LIN {X 0,Y 291.484,Z 681.746,A -85,B 0,C 180,E1 17047.292,E2 17047.292} C_VEL
LIN {X 0,Y 289.004,Z 660.075,A -85,B 0,C 180,E1 17052.26,E2 17052.26} C_VEL
LIN {X 0,Y 282.75,Z 637.12,A -85,B 0,C 180,E1 17057.64,E2 17057.64} C_VEL
LIN {X 0,Y 273.283,Z 615.443,A -85,B 0,C 180,E1 17063.436,E2 17063.436} C_VEL
LIN {X 0,Y 264.026,Z 599.669,A -85,B 0,C 180,E1 17068.648,E2 17068.648} C_VEL
LIN {X 0,Y 259.999,Z 593.567,A -85,B 0,C 180,E1 17071.016,E2 17071.016} C_VEL
LIN {X 0,Y 256.449,Z 587.64,A -85,B 0,C 180,E1 17073.314,E2 17073.314} C_VEL
LIN {X 0,Y 252.817,Z 583.048,A -85,B 0,C 180,E1 17075.688,E2 17075.688} C_VEL
LIN {X 0,Y 252.498,Z 580.66,A -85,B 0,C 180,E1 17076.137,E2 17076.137} C_VEL
LIN {X 0,Y 252.926,Z 580.66,A -85,B 0,C 180,E1 17083.299,E2 17083.299} C_VEL
LIN {X 0,Y 253.73,Z 580.66,A -85,B 0,C 180,E1 17093.136,E2 17093.136} C_VEL
LIN {X 0,Y 254.478,Z 580.66,A -85,B 0,C 180,E1 17099.99,E2 17099.99} C_VEL
LIN {X 0,Y 253.769,Z 580.66,A -85,B 0,C 180,E1 17106.843,E2 17106.843} C_VEL
LIN {X 0,Y 253.149,Z 580.66,A -85,B 0,C 180,E1 17113.831,E2 17113.831} C_VEL
LIN {X 0,Y 252.816,Z 580.66,A -85,B 0,C 180,E1 17117.976,E2 17117.976} C_VEL
LIN {X 0,Y 254.454,Z 585.604,A -85,B 0,C 180,E1 17119.318,E2 17119.318} C_VEL
LIN {X 0,Y 258.108,Z 589.393,A -85,B 0,C 180,E1 17121.472,E2 17121.472} C_VEL
LIN {X 0,Y 268.336,Z 604.22,A -85,B 0,C 180,E1 17126.709,E2 17126.709} C_VEL
LIN {X 0,Y 281.648,Z 625.679,A -85,B 0,C 180,E1 17132.393,E2 17132.393} C_VEL
LIN {X 0,Y 293.764,Z 651.604,A -85,B 0,C 180,E1 17137.493,E2 17137.493} C_VEL
LIN {X 0,Y 302.264,Z 679.148,A -85,B 0,C 180,E1 17141.931,E2 17141.931} C_VEL
LIN {X 0,Y 292.999,Z 713.963,A -85,B 0,C 180,E1 17144.982,E2 17144.982} C_VEL
LIN {X 0,Y 282.558,Z 745.546,A -85,B 0,C 180,E1 17149.094,E2 17149.094} C_VEL
LIN {X 0,Y 272.431,Z 773.196,A -85,B 0,C 180,E1 17154.352,E2 17154.352} C_VEL
LIN {X 0,Y 264.031,Z 796.979,A -85,B 0,C 180,E1 17160.826,E2 17160.826} C_VEL
LIN {X 0,Y 258.28,Z 816.418,A -85,B 0,C 180,E1 17168.505,E2 17168.505} C_VEL
LIN {X 0,Y 256.334,Z 829.468,A -85,B 0,C 180,E1 17176.331,E2 17176.331} C_VEL
LIN {X 0,Y 256.467,Z 836.245,A -85,B 0,C 180,E1 17183.216,E2 17183.216} C_VEL
LIN {X 0,Y 256.973,Z 838.591,A -85,B 0,C 180,E1 17189.997,E2 17189.997} C_VEL
LIN {X 0,Y 256.471,Z 836.262,A -85,B 0,C 180,E1 17196.777,E2 17196.777} C_VEL
LIN {X 0,Y 256.43,Z 828.378,A -85,B 0,C 180,E1 17204.529,E2 17204.529} C_VEL
LIN {X 0,Y 258.845,Z 814.689,A -85,B 0,C 180,E1 17212.342,E2 17212.342} C_VEL
LIN {X 0,Y 264.923,Z 794.449,A -85,B 0,C 180,E1 17220,E2 17220} C_VEL
LIN {X 0,Y 273.864,Z 769.676,A -85,B 0,C 180,E1 17226.456,E2 17226.456} C_VEL
LIN {X 0,Y 284.359,Z 740.416,A -85,B 0,C 180,E1 17231.705,E2 17231.705} C_VEL
LIN {X 0,Y 294.985,Z 707.872,A -85,B 0,C 180,E1 17235.668,E2 17235.668} C_VEL
LIN {X 0,Y 302.325,Z 679.287,A -85,B 0,C 180,E1 17238.079,E2 17238.079} C_VEL
LIN {X 0,Y 293.689,Z 651.111,A -85,B 0,C 180,E1 17242.612,E2 17242.612} C_VEL
LIN {X 0,Y 281.361,Z 624.993,A -85,B 0,C 180,E1 17247.798,E2 17247.798} C_VEL
LIN {X 0,Y 266.547,Z 601.233,A -85,B 0,C 180,E1 17254.232,E2 17254.232} C_VEL
LIN {X 0,Y 260.669,Z 593.537,A -85,B 0,C 180,E1 17257.169,E2 17257.169} C_VEL
LIN {X 0,Y 257.32,Z 587.873,A -85,B 0,C 180,E1 17259.141,E2 17259.141} C_VEL
LIN {X 0,Y 248.734,Z 587.348,A -85,B 0,C 180,E1 17264.144,E2 17264.144} C_VEL
LIN {X 0,Y 245.41,Z 582.419,A -85,B 0,C 180,E1 17267.087,E2 17267.087} C_VEL
LIN {X 0,Y 245.226,Z 580.66,A -85,B 0,C 180,E1 17267.531,E2 17267.531} C_VEL
LIN {X 0,Y 246.174,Z 580.66,A -85,B 0,C 180,E1 17276.484,E2 17276.484} C_VEL
LIN {X 0,Y 246.571,Z 580.66,A -85,B 0,C 180,E1 17280.01,E2 17280.01} C_VEL
LIN {X 0,Y 245.547,Z 580.66,A -85,B 0,C 180,E1 17289.43,E2 17289.43} C_VEL
LIN {X 0,Y 244.844,Z 580.933,A -85,B 0,C 180,E1 17298.253,E2 17298.253} C_VEL
LIN {X 0,Y 246.48,Z 585.654,A -85,B 0,C 180,E1 17300.107,E2 17300.107} C_VEL
LIN {X 0,Y 250.248,Z 588.949,A -85,B 0,C 180,E1 17303.05,E2 17303.05} C_VEL
LIN {X 0,Y 253.602,Z 594.604,A -85,B 0,C 180,E1 17305.659,E2 17305.659} C_VEL
LIN {X 0,Y 260.13,Z 605.185,A -85,B 0,C 180,E1 17310.114,E2 17310.114} C_VEL
LIN {X 0,Y 268.683,Z 620.445,A -85,B 0,C 180,E1 17315.49,E2 17315.49} C_VEL
LIN {X 0,Y 277.671,Z 642.456,A -85,B 0,C 180,E1 17321.657,E2 17321.657} C_VEL
LIN {X 0,Y 283.118,Z 664.136,A -85,B 0,C 180,E1 17327.005,E2 17327.005} C_VEL
LIN {X 0,Y 284.976,Z 686.052,A -85,B 0,C 180,E1 17332.261,E2 17332.261} C_VEL
LIN {X 0,Y 282.565,Z 694.344,A -85,B 0,C 180,E1 17333.89,E2 17333.89} C_VEL
LIN {X 0,Y 272.426,Z 717.171,A -85,B 0,C 180,E1 17339.068,E2 17339.068} C_VEL
LIN {X 0,Y 263.2,Z 735.869,A -85,B 0,C 180,E1 17345.355,E2 17345.355} C_VEL
LIN {X 0,Y 255.905,Z 749.866,A -85,B 0,C 180,E1 17352.797,E2 17352.797} C_VEL
LIN {X 0,Y 252.105,Z 757.453,A -85,B 0,C 180,E1 17359.624,E2 17359.624} C_VEL
LIN {X 0,Y 250.5,Z 761.052,A -85,B 0,C 180,E1 17366.538,E2 17366.538} C_VEL
LIN {X 0,Y 250.561,Z 761.007,A -85,B 0,C 180,E1 17373.467,E2 17373.467} C_VEL
LIN {X 0,Y 252.885,Z 755.837,A -85,B 0,C 180,E1 17382.099,E2 17382.099} C_VEL
LIN {X 0,Y 258.292,Z 745.196,A -85,B 0,C 180,E1 17390.003,E2 17390.003} C_VEL
LIN {X 0,Y 266.486,Z 729.264,A -85,B 0,C 180,E1 17397.037,E2 17397.037} C_VEL
LIN {X 0,Y 276.708,Z 707.849,A -85,B 0,C 180,E1 17403.175,E2 17403.175} C_VEL
LIN {X 0,Y 284.948,Z 687.938,A -85,B 0,C 180,E1 17407.141,E2 17407.141} C_VEL
LIN {X 0,Y 283.223,Z 665.7,A -85,B 0,C 180,E1 17412.51,E2 17412.51} C_VEL
LIN {X 0,Y 278.054,Z 643.824,A -85,B 0,C 180,E1 17417.844,E2 17417.844} C_VEL
LIN {X 0,Y 269.633,Z 622.585,A -85,B 0,C 180,E1 17423.715,E2 17423.715} C_VEL
LIN {X 0,Y 260.505,Z 605.867,A -85,B 0,C 180,E1 17429.442,E2 17429.442} C_VEL
LIN {X 0,Y 253.604,Z 594.637,A -85,B 0,C 180,E1 17434.104,E2 17434.104} C_VEL
LIN {X 0,Y 250.213,Z 589.003,A -85,B 0,C 180,E1 17436.711,E2 17436.711} C_VEL
LIN {X 0,Y 245.039,Z 582.819,A -85,B 0,C 180,E1 17441.061,E2 17441.061} C_VEL
LIN {X 0,Y 244.819,Z 580.66,A -85,B 0,C 180,E1 17441.745,E2 17441.745} C_VEL
LIN {X 0,Y 245.509,Z 580.66,A -85,B 0,C 180,E1 17450.663,E2 17450.663} C_VEL
LIN {X 0,Y 246.202,Z 580.66,A -85,B 0,C 180,E1 17456.465,E2 17456.465} C_VEL
LIN {X 0,Y 246.568,Z 580.66,A -85,B 0,C 180,E1 17459.99,E2 17459.99} C_VEL
LIN {X 0,Y 245.554,Z 580.66,A -85,B 0,C 180,E1 17469.4,E2 17469.4} C_VEL
LIN {X 0,Y 245.295,Z 581.397,A -85,B 0,C 180,E1 17472.919,E2 17472.919} C_VEL
LIN {X 0,Y 247.819,Z 586.604,A -85,B 0,C 180,E1 17475.335,E2 17475.335} C_VEL
LIN {X 0,Y 250.708,Z 589.38,A -85,B 0,C 180,E1 17477.455,E2 17477.455} C_VEL
LIN {X 0,Y 254.799,Z 594.985,A -85,B 0,C 180,E1 17480.195,E2 17480.195} C_VEL
LIN {X 0,Y 265.726,Z 611.439,A -85,B 0,C 180,E1 17486.194,E2 17486.194} C_VEL
LIN {X 0,Y 277.92,Z 632.265,A -85,B 0,C 180,E1 17491.843,E2 17491.843} C_VEL
LIN {X 0,Y 288.974,Z 657.419,A -85,B 0,C 180,E1 17496.988,E2 17496.988} C_VEL
LIN {X 0,Y 295.98,Z 681.869,A -85,B 0,C 180,E1 17501.112,E2 17501.112} C_VEL
LIN {X 0,Y 285.816,Z 717.211,A -85,B 0,C 180,E1 17504.343,E2 17504.343} C_VEL
LIN {X 0,Y 274.522,Z 749.194,A -85,B 0,C 180,E1 17508.821,E2 17508.821} C_VEL
LIN {X 0,Y 263.808,Z 777.218,A -85,B 0,C 180,E1 17514.59,E2 17514.59} C_VEL
LIN {X 0,Y 255.114,Z 800.615,A -85,B 0,C 180,E1 17521.652,E2 17521.652} C_VEL
LIN {X 0,Y 249.861,Z 818.715,A -85,B 0,C 180,E1 17529.658,E2 17529.658} C_VEL
LIN {X 0,Y 248.446,Z 829.786,A -85,B 0,C 180,E1 17537.128,E2 17537.128} C_VEL
LIN {X 0,Y 248.614,Z 835.043,A -85,B 0,C 180,E1 17543.001,E2 17543.001} C_VEL
LIN {X 0,Y 249.15,Z 837.403,A -85,B 0,C 180,E1 17549.997,E2 17549.997} C_VEL
LIN {X 0,Y 248.62,Z 835.06,A -85,B 0,C 180,E1 17556.992,E2 17556.992} C_VEL
LIN {X 0,Y 248.614,Z 827.147,A -85,B 0,C 180,E1 17564.997,E2 17564.997} C_VEL
LIN {X 0,Y 251.283,Z 813.429,A -85,B 0,C 180,E1 17573.053,E2 17573.053} C_VEL
LIN {X 0,Y 257.823,Z 793.166,A -85,B 0,C 180,E1 17580.915,E2 17580.915} C_VEL
LIN {X 0,Y 267.53,Z 767.817,A -85,B 0,C 180,E1 17587.614,E2 17587.614} C_VEL
LIN {X 0,Y 278.305,Z 739.048,A -85,B 0,C 180,E1 17592.825,E2 17592.825} C_VEL
LIN {X 0,Y 289.404,Z 706.392,A -85,B 0,C 180,E1 17596.81,E2 17596.81} C_VEL
LIN {X 0,Y 295.831,Z 680.996,A -85,B 0,C 180,E1 17599.06,E2 17599.06} C_VEL
LIN {X 0,Y 287.805,Z 654.157,A -85,B 0,C 180,E1 17603.663,E2 17603.663} C_VEL
LIN {X 0,Y 276.684,Z 629.753,A -85,B 0,C 180,E1 17608.803,E2 17608.803} C_VEL
LIN {X 0,Y 263.656,Z 607.901,A -85,B 0,C 180,E1 17614.954,E2 17614.954} C_VEL
LIN {X 0,Y 254.144,Z 594.536,A -85,B 0,C 180,E1 17620.318,E2 17620.318} C_VEL
LIN {X 0,Y 250.515,Z 588.746,A -85,B 0,C 180,E1 17622.875,E2 17622.875} C_VEL
LIN {X 0,Y 248.734,Z 587.348,A -85,B 0,C 180,E1 17624.144,E2 17624.144} C_VEL
LIN {X 0,Y 242.06,Z 587.782,A -85,B 0,C 180,E1 17629.455,E2 17629.455} C_VEL
LIN {X 0,Y 238.235,Z 582.554,A -85,B 0,C 180,E1 17635.111,E2 17635.111} C_VEL
LIN {X 0,Y 238.155,Z 580.66,A -85,B 0,C 180,E1 17635.909,E2 17635.909} C_VEL
LIN {X 0,Y 238.66,Z 580.66,A -85,B 0,C 180,E1 17640.01,E2 17640.01} C_VEL
LIN {X 0,Y 237.666,Z 581.2,A -85,B 0,C 180,E1 17649.443,E2 17649.443} C_VEL
LIN {X 0,Y 239.854,Z 586.504,A -85,B 0,C 180,E1 17653.936,E2 17653.936} C_VEL
LIN {X 0,Y 243.016,Z 589.19,A -85,B 0,C 180,E1 17657.679,E2 17657.679} C_VEL
LIN {X 0,Y 246.273,Z 594.62,A -85,B 0,C 180,E1 17661.044,E2 17661.044} C_VEL
LIN {X 0,Y 248.141,Z 596.956,A -85,B 0,C 180,E1 17662.664,E2 17662.664} C_VEL
LIN {X 0,Y 256.047,Z 609.94,A -85,B 0,C 180,E1 17668.846,E2 17668.846} C_VEL
LIN {X 0,Y 265.703,Z 629.267,A -85,B 0,C 180,E1 17675.749,E2 17675.749} C_VEL
LIN {X 0,Y 273.446,Z 651.309,A -85,B 0,C 180,E1 17682.026,E2 17682.026} C_VEL
LIN {X 0,Y 277.677,Z 672.925,A -85,B 0,C 180,E1 17687.564,E2 17687.564} C_VEL
LIN {X 0,Y 277.956,Z 691.579,A -85,B 0,C 180,E1 17692.207,E2 17692.207} C_VEL
LIN {X 0,Y 267.183,Z 715.618,A -85,B 0,C 180,E1 17697.434,E2 17697.434} C_VEL
LIN {X 0,Y 257.196,Z 735.039,A -85,B 0,C 180,E1 17703.804,E2 17703.804} C_VEL
LIN {X 0,Y 249.54,Z 749.077,A -85,B 0,C 180,E1 17710.885,E2 17710.885} C_VEL
LIN {X 0,Y 244.43,Z 758.639,A -85,B 0,C 180,E1 17719.294,E2 17719.294} C_VEL
LIN {X 0,Y 242.708,Z 762.238,A -85,B 0,C 180,E1 17726.427,E2 17726.427} C_VEL
LIN {X 0,Y 242.76,Z 762.195,A -85,B 0,C 180,E1 17733.579,E2 17733.579} C_VEL
LIN {X 0,Y 245.265,Z 757.026,A -85,B 0,C 180,E1 17742.481,E2 17742.481} C_VEL
LIN {X 0,Y 250.964,Z 746.39,A -85,B 0,C 180,E1 17750.613,E2 17750.613} C_VEL
LIN {X 0,Y 259.539,Z 730.479,A -85,B 0,C 180,E1 17757.822,E2 17757.822} C_VEL
LIN {X 0,Y 270.224,Z 709.091,A -85,B 0,C 180,E1 17764.079,E2 17764.079} C_VEL
LIN {X 0,Y 278.32,Z 689.31,A -85,B 0,C 180,E1 17768.182,E2 17768.182} C_VEL
LIN {X 0,Y 276.857,Z 667.842,A -85,B 0,C 180,E1 17773.59,E2 17773.59} C_VEL
LIN {X 0,Y 271.994,Z 646.383,A -85,B 0,C 180,E1 17779.127,E2 17779.127} C_VEL
LIN {X 0,Y 264.392,Z 626.168,A -85,B 0,C 180,E1 17785.054,E2 17785.054} C_VEL
LIN {X 0,Y 254.755,Z 607.962,A -85,B 0,C 180,E1 17791.849,E2 17791.849} C_VEL
LIN {X 0,Y 250.273,Z 600.944,A -85,B 0,C 180,E1 17795.247,E2 17795.247} C_VEL
LIN {X 0,Y 246.888,Z 595.127,A -85,B 0,C 180,E1 17798.164,E2 17798.164} C_VEL
LIN {X 0,Y 243.091,Z 589.722,A -85,B 0,C 180,E1 17801.845,E2 17801.845} C_VEL
LIN {X 0,Y 242.171,Z 588.089,A -85,B 0,C 180,E1 17802.907,E2 17802.907} C_VEL
LIN {X 0,Y 237.857,Z 583.161,A -85,B 0,C 180,E1 17809.067,E2 17809.067} C_VEL
LIN {X 0,Y 237.594,Z 580.66,A -85,B 0,C 180,E1 17810.349,E2 17810.349} C_VEL
LIN {X 0,Y 238.273,Z 580.66,A -85,B 0,C 180,E1 17816.347,E2 17816.347} C_VEL
LIN {X 0,Y 238.657,Z 580.66,A -85,B 0,C 180,E1 17819.99,E2 17819.99} C_VEL
LIN {X 0,Y 238.09,Z 581.405,A -85,B 0,C 180,E1 17824.892,E2 17824.892} C_VEL
LIN {X 0,Y 240.232,Z 586.467,A -85,B 0,C 180,E1 17828.716,E2 17828.716} C_VEL
LIN {X 0,Y 243.552,Z 589.301,A -85,B 0,C 180,E1 17832.329,E2 17832.329} C_VEL
LIN {X 0,Y 247.027,Z 594.819,A -85,B 0,C 180,E1 17835.544,E2 17835.544} C_VEL
LIN {X 0,Y 248.92,Z 597.304,A -85,B 0,C 180,E1 17837.01,E2 17837.01} C_VEL
LIN {X 0,Y 254.727,Z 605.939,A -85,B 0,C 180,E1 17840.997,E2 17840.997} C_VEL
LIN {X 0,Y 263.523,Z 619.355,A -85,B 0,C 180,E1 17845.971,E2 17845.971} C_VEL
LIN {X 0,Y 275.76,Z 642.16,A -85,B 0,C 180,E1 17852.122,E2 17852.122} C_VEL
LIN {X 0,Y 285.4,Z 667.461,A -85,B 0,C 180,E1 17857.271,E2 17857.271} C_VEL
LIN {X 0,Y 289.633,Z 684.994,A -85,B 0,C 180,E1 17860.282,E2 17860.282} C_VEL
LIN {X 0,Y 278.654,Z 720.111,A -85,B 0,C 180,E1 17863.667,E2 17863.667} C_VEL
LIN {X 0,Y 267.152,Z 751.162,A -85,B 0,C 180,E1 17868.244,E2 17868.244} C_VEL
LIN {X 0,Y 255.963,Z 778.674,A -85,B 0,C 180,E1 17874.256,E2 17874.256} C_VEL
LIN {X 0,Y 247.441,Z 800.68,A -85,B 0,C 180,E1 17881.252,E2 17881.252} C_VEL
LIN {X 0,Y 241.917,Z 818.856,A -85,B 0,C 180,E1 17889.817,E2 17889.817} C_VEL
LIN {X 0,Y 240.556,Z 829.8,A -85,B 0,C 180,E1 17897.908,E2 17897.908} C_VEL
LIN {X 0,Y 240.76,Z 833.839,A -85,B 0,C 180,E1 17902.771,E2 17902.771} C_VEL
LIN {X 0,Y 241.326,Z 836.214,A -85,B 0,C 180,E1 17909.997,E2 17909.997} C_VEL
LIN {X 0,Y 240.766,Z 833.858,A -85,B 0,C 180,E1 17917.222,E2 17917.222} C_VEL
LIN {X 0,Y 240.804,Z 825.915,A -85,B 0,C 180,E1 17925.495,E2 17925.495} C_VEL
LIN {X 0,Y 243.72,Z 812.161,A -85,B 0,C 180,E1 17933.812,E2 17933.812} C_VEL
LIN {X 0,Y 250.713,Z 792.046,A -85,B 0,C 180,E1 17941.83,E2 17941.83} C_VEL
LIN {X 0,Y 261.116,Z 766.508,A -85,B 0,C 180,E1 17948.706,E2 17948.706} C_VEL
LIN {X 0,Y 272.271,Z 737.882,A -85,B 0,C 180,E1 17953.966,E2 17953.966} C_VEL
LIN {X 0,Y 283.902,Z 704.895,A -85,B 0,C 180,E1 17958.007,E2 17958.007} C_VEL
LIN {X 0,Y 289.587,Z 683.6,A -85,B 0,C 180,E1 17959.943,E2 17959.943} C_VEL
LIN {X 0,Y 282.141,Z 657.535,A -85,B 0,C 180,E1 17964.653,E2 17964.653} C_VEL
LIN {X 0,Y 271.947,Z 634.447,A -85,B 0,C 180,E1 17969.825,E2 17969.825} C_VEL
LIN {X 0,Y 260.53,Z 614.345,A -85,B 0,C 180,E1 17975.779,E2 17975.779} C_VEL
LIN {X 0,Y 251.677,Z 601.43,A -85,B 0,C 180,E1 17981.145,E2 17981.145} C_VEL
LIN {X 0,Y 247.246,Z 594.982,A -85,B 0,C 180,E1 17984.47,E2 17984.47} C_VEL
LIN {X 0,Y 243.547,Z 589.353,A -85,B 0,C 180,E1 17987.899,E2 17987.899} C_VEL
LIN {X 0,Y 242.06,Z 587.782,A -85,B 0,C 180,E1 17989.455,E2 17989.455} C_VEL
LIN {X 0,Y 236.289,Z 588.291,A -85,B 0,C 180,E1 17997.671,E2 17997.671} C_VEL
LIN {X 0,Y 236.476,Z 589.167,A -85,B 0,C 180,E1 18009.071,E2 18009.071} C_VEL
LIN {X 0,Y 239.066,Z 594.704,A -85,B 0,C 180,E1 18014.45,E2 18014.45} C_VEL
LIN {X 0,Y 241.246,Z 597.021,A -85,B 0,C 180,E1 18017.26,E2 18017.26} C_VEL
LIN {X 0,Y 244.913,Z 602.642,A -85,B 0,C 180,E1 18021.232,E2 18021.232} C_VEL
LIN {X 0,Y 252.764,Z 616.714,A -85,B 0,C 180,E1 18028.277,E2 18028.277} C_VEL
LIN {X 0,Y 261.635,Z 635.872,A -85,B 0,C 180,E1 18035.369,E2 18035.369} C_VEL
LIN {X 0,Y 268.096,Z 656.605,A -85,B 0,C 180,E1 18041.522,E2 18041.522} C_VEL
LIN {X 0,Y 271.517,Z 677.591,A -85,B 0,C 180,E1 18047.151,E2 18047.151} C_VEL
LIN {X 0,Y 271.508,Z 693.613,A -85,B 0,C 180,E1 18051.338,E2 18051.338} C_VEL
LIN {X 0,Y 259.89,Z 718.23,A -85,B 0,C 180,E1 18056.9,E2 18056.9} C_VEL
LIN {X 0,Y 249.089,Z 738.273,A -85,B 0,C 180,E1 18063.857,E2 18063.857} C_VEL
LIN {X 0,Y 240.981,Z 752.253,A -85,B 0,C 180,E1 18071.695,E2 18071.695} C_VEL
LIN {X 0,Y 236.751,Z 759.827,A -85,B 0,C 180,E1 18078.943,E2 18078.943} C_VEL
LIN {X 0,Y 234.93,Z 763.421,A -85,B 0,C 180,E1 18086.308,E2 18086.308} C_VEL
LIN {X 0,Y 234.981,Z 763.379,A -85,B 0,C 180,E1 18093.698,E2 18093.698} C_VEL
LIN {X 0,Y 237.624,Z 758.219,A -85,B 0,C 180,E1 18102.889,E2 18102.889} C_VEL
LIN {X 0,Y 243.553,Z 747.763,A -85,B 0,C 180,E1 18111.151,E2 18111.151} C_VEL
LIN {X 0,Y 252.664,Z 731.689,A -85,B 0,C 180,E1 18118.648,E2 18118.648} C_VEL
LIN {X 0,Y 263.805,Z 710.331,A -85,B 0,C 180,E1 18125.028,E2 18125.028} C_VEL
LIN {X 0,Y 271.698,Z 692.758,A -85,B 0,C 180,E1 18128.712,E2 18128.712} C_VEL
LIN {X 0,Y 270.897,Z 672.694,A -85,B 0,C 180,E1 18134.023,E2 18134.023} C_VEL
LIN {X 0,Y 266.687,Z 651.162,A -85,B 0,C 180,E1 18139.858,E2 18139.858} C_VEL
LIN {X 0,Y 260.015,Z 631.997,A -85,B 0,C 180,E1 18145.728,E2 18145.728} C_VEL
LIN {X 0,Y 251.413,Z 614.593,A -85,B 0,C 180,E1 18152.533,E2 18152.533} C_VEL
LIN {X 0,Y 246.97,Z 607.143,A -85,B 0,C 180,E1 18156.315,E2 18156.315} C_VEL
LIN {X 0,Y 244.314,Z 602.206,A -85,B 0,C 180,E1 18158.992,E2 18158.992} C_VEL
LIN {X 0,Y 240.973,Z 596.177,A -85,B 0,C 180,E1 18162.801,E2 18162.801} C_VEL
LIN {X 0,Y 236.532,Z 590.526,A -85,B 0,C 180,E1 18169.674,E2 18169.674} C_VEL
LIN {X 0,Y 236.148,Z 588.418,A -85,B 0,C 180,E1 18171.167,E2 18171.167} C_VEL
LIN {X 0,Y 236.756,Z 588.624,A -85,B 0,C 180,E1 18184.115,E2 18184.115} C_VEL
LIN {X 0,Y 239.158,Z 594.317,A -85,B 0,C 180,E1 18188.637,E2 18188.637} C_VEL
LIN {X 0,Y 241.971,Z 597.044,A -85,B 0,C 180,E1 18191.837,E2 18191.837} C_VEL
LIN {X 0,Y 245.968,Z 602.77,A -85,B 0,C 180,E1 18195.612,E2 18195.612} C_VEL
LIN {X 0,Y 255.448,Z 617.73,A -85,B 0,C 180,E1 18202.419,E2 18202.419} C_VEL
LIN {X 0,Y 266.117,Z 636.709,A -85,B 0,C 180,E1 18208.561,E2 18208.561} C_VEL
LIN {X 0,Y 275.962,Z 659.496,A -85,B 0,C 180,E1 18214.058,E2 18214.058} C_VEL
LIN {X 0,Y 283.36,Z 686.138,A -85,B 0,C 180,E1 18219.182,E2 18219.182} C_VEL
LIN {X 0,Y 272.532,Z 720.298,A -85,B 0,C 180,E1 18222.63,E2 18222.63} C_VEL
LIN {X 0,Y 260.217,Z 751.913,A -85,B 0,C 180,E1 18227.435,E2 18227.435} C_VEL
LIN {X 0,Y 248.678,Z 778.946,A -85,B 0,C 180,E1 18233.583,E2 18233.583} C_VEL
LIN {X 0,Y 239.535,Z 801.306,A -85,B 0,C 180,E1 18241.051,E2 18241.051} C_VEL
LIN {X 0,Y 234.224,Z 817.599,A -85,B 0,C 180,E1 18249.123,E2 18249.123} C_VEL
LIN {X 0,Y 232.69,Z 828.457,A -85,B 0,C 180,E1 18257.373,E2 18257.373} C_VEL
LIN {X 0,Y 232.906,Z 832.636,A -85,B 0,C 180,E1 18262.526,E2 18262.526} C_VEL
LIN {X 0,Y 233.501,Z 835.026,A -85,B 0,C 180,E1 18269.997,E2 18269.997} C_VEL
LIN {X 0,Y 232.914,Z 832.656,A -85,B 0,C 180,E1 18277.467,E2 18277.467} C_VEL
LIN {X 0,Y 233.013,Z 824.682,A -85,B 0,C 180,E1 18286.027,E2 18286.027} C_VEL
LIN {X 0,Y 236.213,Z 810.896,A -85,B 0,C 180,E1 18294.618,E2 18294.618} C_VEL
LIN {X 0,Y 243.79,Z 790.821,A -85,B 0,C 180,E1 18302.828,E2 18302.828} C_VEL
LIN {X 0,Y 254.627,Z 765.428,A -85,B 0,C 180,E1 18309.813,E2 18309.813} C_VEL
LIN {X 0,Y 266.467,Z 736.529,A -85,B 0,C 180,E1 18315.181,E2 18315.181} C_VEL
LIN {X 0,Y 278.26,Z 704.396,A -85,B 0,C 180,E1 18319.146,E2 18319.146} C_VEL
LIN {X 0,Y 283.398,Z 686.418,A -85,B 0,C 180,E1 18320.816,E2 18320.816} C_VEL
LIN {X 0,Y 276.553,Z 660.888,A -85,B 0,C 180,E1 18325.689,E2 18325.689} C_VEL
LIN {X 0,Y 266.944,Z 638.252,A -85,B 0,C 180,E1 18331.072,E2 18331.072} C_VEL
LIN {X 0,Y 256.73,Z 619.872,A -85,B 0,C 180,E1 18336.897,E2 18336.897} C_VEL
LIN {X 0,Y 249.144,Z 608.232,A -85,B 0,C 180,E1 18341.979,E2 18341.979} C_VEL
LIN {X 0,Y 245.37,Z 602.346,A -85,B 0,C 180,E1 18345.036,E2 18345.036} C_VEL
LIN {X 0,Y 241.741,Z 596.221,A -85,B 0,C 180,E1 18348.723,E2 18348.723} C_VEL
LIN {X 0,Y 237.07,Z 590.392,A -85,B 0,C 180,E1 18355.431,E2 18355.431} C_VEL
LIN {X 0,Y 236.448,Z 588.331,A -85,B 0,C 180,E1 18357.258,E2 18357.258} C_VEL
LIN {X 0,Y 236.289,Z 588.291,A -85,B 0,C 180,E1 18357.671,E2 18357.671} C_VEL
LIN {X 0,Y 234.846,Z 591.965,A -85,B 0,C 180,E1 18361.814,E2 18361.814} C_VEL
LIN {X 0,Y 234.493,Z 596.014,A -85,B 0,C 180,E1 18365.988,E2 18365.988} C_VEL
LIN {X 0,Y 235.214,Z 597.29,A -85,B 0,C 180,E1 18368.902,E2 18368.902} C_VEL
LIN {X 0,Y 237.932,Z 602.797,A -85,B 0,C 180,E1 18374.951,E2 18374.951} C_VEL
LIN {X 0,Y 239.408,Z 605.1,A -85,B 0,C 180,E1 18377.049,E2 18377.049} C_VEL
LIN {X 0,Y 243.461,Z 612.242,A -85,B 0,C 180,E1 18381.919,E2 18381.919} C_VEL
LIN {X 0,Y 249.259,Z 623.12,A -85,B 0,C 180,E1 18387.602,E2 18387.602} C_VEL
LIN {X 0,Y 257.37,Z 642.395,A -85,B 0,C 180,E1 18395.01,E2 18395.01} C_VEL
LIN {X 0,Y 263.088,Z 663.82,A -85,B 0,C 180,E1 18401.576,E2 18401.576} C_VEL
LIN {X 0,Y 265.468,Z 684.446,A -85,B 0,C 180,E1 18407.344,E2 18407.344} C_VEL
LIN {X 0,Y 264.76,Z 696.526,A -85,B 0,C 180,E1 18410.594,E2 18410.594} C_VEL
LIN {X 0,Y 252.628,Z 720.834,A -85,B 0,C 180,E1 18416.337,E2 18416.337} C_VEL
LIN {X 0,Y 242.086,Z 739.476,A -85,B 0,C 180,E1 18423.04,E2 18423.04} C_VEL
LIN {X 0,Y 233.555,Z 753.447,A -85,B 0,C 180,E1 18431.091,E2 18431.091} C_VEL
LIN {X 0,Y 229.082,Z 761.015,A -85,B 0,C 180,E1 18438.568,E2 18438.568} C_VEL
LIN {X 0,Y 227.158,Z 764.604,A -85,B 0,C 180,E1 18446.182,E2 18446.182} C_VEL
LIN {X 0,Y 227.187,Z 764.566,A -85,B 0,C 180,E1 18453.825,E2 18453.825} C_VEL
LIN {X 0,Y 230.007,Z 759.409,A -85,B 0,C 180,E1 18463.323,E2 18463.323} C_VEL
LIN {X 0,Y 236.265,Z 748.959,A -85,B 0,C 180,E1 18471.836,E2 18471.836} C_VEL
LIN {X 0,Y 245.824,Z 732.904,A -85,B 0,C 180,E1 18479.523,E2 18479.523} C_VEL
LIN {X 0,Y 257.452,Z 711.57,A -85,B 0,C 180,E1 18486.025,E2 18486.025} C_VEL
LIN {X 0,Y 265.19,Z 694.135,A -85,B 0,C 180,E1 18489.848,E2 18489.848} C_VEL
LIN {X 0,Y 264.585,Z 674.128,A -85,B 0,C 180,E1 18495.385,E2 18495.385} C_VEL
LIN {X 0,Y 260.672,Z 653.388,A -85,B 0,C 180,E1 18501.352,E2 18501.352} C_VEL
LIN {X 0,Y 254.264,Z 634.706,A -85,B 0,C 180,E1 18507.583,E2 18507.583} C_VEL
LIN {X 0,Y 245.938,Z 616.464,A -85,B 0,C 180,E1 18515.315,E2 18515.315} C_VEL
LIN {X 0,Y 241.539,Z 609.13,A -85,B 0,C 180,E1 18519.826,E2 18519.826} C_VEL
LIN {X 0,Y 238.359,Z 603.169,A -85,B 0,C 180,E1 18524.075,E2 18524.075} C_VEL
LIN {X 0,Y 235.103,Z 597.709,A -85,B 0,C 180,E1 18530.417,E2 18530.417} C_VEL
LIN {X 0,Y 234.697,Z 596.131,A -85,B 0,C 180,E1 18532.021,E2 18532.021} C_VEL
LIN {X 0,Y 235.482,Z 596.488,A -85,B 0,C 180,E1 18543.676,E2 18543.676} C_VEL
LIN {X 0,Y 238.555,Z 602.693,A -85,B 0,C 180,E1 18549.349,E2 18549.349} C_VEL
LIN {X 0,Y 240.442,Z 605.051,A -85,B 0,C 180,E1 18551.568,E2 18551.568} C_VEL
LIN {X 0,Y 245.157,Z 612.751,A -85,B 0,C 180,E1 18556.24,E2 18556.24} C_VEL
LIN {X 0,Y 252.377,Z 624.173,A -85,B 0,C 180,E1 18561.663,E2 18561.663} C_VEL
LIN {X 0,Y 262.542,Z 643.595,A -85,B 0,C 180,E1 18568.141,E2 18568.141} C_VEL
LIN {X 0,Y 271.647,Z 666.876,A -85,B 0,C 180,E1 18573.862,E2 18573.862} C_VEL
LIN {X 0,Y 277.054,Z 688.498,A -85,B 0,C 180,E1 18578.198,E2 18578.198} C_VEL
LIN {X 0,Y 265.974,Z 721.928,A -85,B 0,C 180,E1 18581.723,E2 18581.723} C_VEL
LIN {X 0,Y 253.346,Z 752.61,A -85,B 0,C 180,E1 18586.583,E2 18586.583} C_VEL
LIN {X 0,Y 241.414,Z 779.216,A -85,B 0,C 180,E1 18592.866,E2 18592.866} C_VEL
LIN {X 0,Y 231.809,Z 801.392,A -85,B 0,C 180,E1 18600.665,E2 18600.665} C_VEL
LIN {X 0,Y 226.193,Z 818.129,A -85,B 0,C 180,E1 18609.539,E2 18609.539} C_VEL
LIN {X 0,Y 224.824,Z 828.563,A -85,B 0,C 180,E1 18618.341,E2 18618.341} C_VEL
LIN {X 0,Y 225.251,Z 833.15,A -85,B 0,C 180,E1 18626.142,E2 18626.142} C_VEL
LIN {X 0,Y 225.693,Z 833.839,A -85,B 0,C 180,E1 18629.996,E2 18629.996} C_VEL
LIN {X 0,Y 225.051,Z 831.45,A -85,B 0,C 180,E1 18637.729,E2 18637.729} C_VEL
LIN {X 0,Y 225.221,Z 823.447,A -85,B 0,C 180,E1 18646.597,E2 18646.597} C_VEL
LIN {X 0,Y 228.788,Z 809.639,A -85,B 0,C 180,E1 18655.473,E2 18655.473} C_VEL
LIN {X 0,Y 236.697,Z 789.969,A -85,B 0,C 180,E1 18663.761,E2 18663.761} C_VEL
LIN {X 0,Y 248.237,Z 764.362,A -85,B 0,C 180,E1 18670.975,E2 18670.975} C_VEL
LIN {X 0,Y 260.886,Z 734.892,A -85,B 0,C 180,E1 18676.497,E2 18676.497} C_VEL
LIN {X 0,Y 273.475,Z 701.54,A -85,B 0,C 180,E1 18680.563,E2 18680.563} C_VEL
LIN {X 0,Y 277.148,Z 688.614,A -85,B 0,C 180,E1 18681.814,E2 18681.814} C_VEL
LIN {X 0,Y 270.718,Z 663.708,A -85,B 0,C 180,E1 18686.872,E2 18686.872} C_VEL
LIN {X 0,Y 262.159,Z 642.794,A -85,B 0,C 180,E1 18692.172,E2 18692.172} C_VEL
LIN {X 0,Y 251.869,Z 622.901,A -85,B 0,C 180,E1 18698.869,E2 18698.869} C_VEL
LIN {X 0,Y 243.253,Z 609.621,A -85,B 0,C 180,E1 18705.709,E2 18705.709} C_VEL
LIN {X 0,Y 239.182,Z 603.072,A -85,B 0,C 180,E1 18710.215,E2 18710.215} C_VEL
LIN {X 0,Y 235.625,Z 597.118,A -85,B 0,C 180,E1 18716.441,E2 18716.441} C_VEL
LIN {X 0,Y 234.572,Z 595.791,A -85,B 0,C 180,E1 18720.01,E2 18720.01} C_VEL
LIN {X 0,Y 234.493,Z 596.014,A -85,B 0,C 180,E1 18725.988,E2 18725.988} C_VEL
LIN {X 0,Y 234.465,Z 599.493,A -85,B 0,C 180,E1 18727.941,E2 18727.941} C_VEL
LIN {X 0,Y 234.076,Z 607.442,A -85,B 0,C 180,E1 18730.656,E2 18730.656} C_VEL
LIN {X 0,Y 234.171,Z 607.839,A -85,B 0,C 180,E1 18731.011,E2 18731.011} C_VEL
LIN {X 0,Y 237.087,Z 612.234,A -85,B 0,C 180,E1 18736.451,E2 18736.451} C_VEL
LIN {X 0,Y 240.824,Z 619.853,A -85,B 0,C 180,E1 18741.652,E2 18741.652} C_VEL
LIN {X 0,Y 246.299,Z 631.438,A -85,B 0,C 180,E1 18747.693,E2 18747.693} C_VEL
LIN {X 0,Y 252.669,Z 648.009,A -85,B 0,C 180,E1 18754.335,E2 18754.335} C_VEL
LIN {X 0,Y 257.475,Z 668.445,A -85,B 0,C 180,E1 18760.902,E2 18760.902} C_VEL
LIN {X 0,Y 259.135,Z 687.764,A -85,B 0,C 180,E1 18766.587,E2 18766.587} C_VEL
LIN {X 0,Y 258.064,Z 699.358,A -85,B 0,C 180,E1 18769.812,E2 18769.812} C_VEL
LIN {X 0,Y 245.373,Z 723.442,A -85,B 0,C 180,E1 18775.738,E2 18775.738} C_VEL
LIN {X 0,Y 233.959,Z 742.504,A -85,B 0,C 180,E1 18783.068,E2 18783.068} C_VEL
LIN {X 0,Y 225.425,Z 755.866,A -85,B 0,C 180,E1 18791.4,E2 18791.4} C_VEL
LIN {X 0,Y 220.659,Z 763.46,A -85,B 0,C 180,E1 18800.127,E2 18800.127} C_VEL
LIN {X 0,Y 219.382,Z 765.788,A -85,B 0,C 180,E1 18806.046,E2 18806.046} C_VEL
LIN {X 0,Y 219.411,Z 765.75,A -85,B 0,C 180,E1 18813.96,E2 18813.96} C_VEL
LIN {X 0,Y 222.393,Z 760.602,A -85,B 0,C 180,E1 18823.788,E2 18823.788} C_VEL
LIN {X 0,Y 228.616,Z 750.793,A -85,B 0,C 180,E1 18832.144,E2 18832.144} C_VEL
LIN {X 0,Y 238.413,Z 735.245,A -85,B 0,C 180,E1 18840.01,E2 18840.01} C_VEL
LIN {X 0,Y 250.367,Z 714.322,A -85,B 0,C 180,E1 18846.671,E2 18846.671} C_VEL
LIN {X 0,Y 258.581,Z 697.735,A -85,B 0,C 180,E1 18850.418,E2 18850.418} C_VEL
LIN {X 0,Y 258.609,Z 678.667,A -85,B 0,C 180,E1 18855.936,E2 18855.936} C_VEL
LIN {X 0,Y 255.593,Z 659.173,A -85,B 0,C 180,E1 18861.797,E2 18861.797} C_VEL
LIN {X 0,Y 249.857,Z 640.253,A -85,B 0,C 180,E1 18868.389,E2 18868.389} C_VEL
LIN {X 0,Y 242.643,Z 623.152,A -85,B 0,C 180,E1 18876.061,E2 18876.061} C_VEL
LIN {X 0,Y 238.722,Z 615.994,A -85,B 0,C 180,E1 18880.659,E2 18880.659} C_VEL
LIN {X 0,Y 235.952,Z 610.472,A -85,B 0,C 180,E1 18884.903,E2 18884.903} C_VEL
LIN {X 0,Y 233.428,Z 604.81,A -85,B 0,C 180,E1 18891.158,E2 18891.158} C_VEL
LIN {X 0,Y 232.644,Z 603.485,A -85,B 0,C 180,E1 18896.258,E2 18896.258} C_VEL
LIN {X 0,Y 234.14,Z 604.781,A -85,B 0,C 180,E1 18903.581,E2 18903.581} C_VEL
LIN {X 0,Y 237.496,Z 610.705,A -85,B 0,C 180,E1 18909.746,E2 18909.746} C_VEL
LIN {X 0,Y 243.052,Z 620.424,A -85,B 0,C 180,E1 18915.92,E2 18915.92} C_VEL
LIN {X 0,Y 249.801,Z 631.987,A -85,B 0,C 180,E1 18921.431,E2 18921.431} C_VEL
LIN {X 0,Y 258.459,Z 649.681,A -85,B 0,C 180,E1 18927.49,E2 18927.49} C_VEL
LIN {X 0,Y 266.518,Z 671.969,A -85,B 0,C 180,E1 18933.183,E2 18933.183} C_VEL
LIN {X 0,Y 270.814,Z 692.585,A -85,B 0,C 180,E1 18937.43,E2 18937.43} C_VEL
LIN {X 0,Y 258.577,Z 725.604,A -85,B 0,C 180,E1 18941.07,E2 18941.07} C_VEL
LIN {X 0,Y 245.55,Z 755.455,A -85,B 0,C 180,E1 18946.112,E2 18946.112} C_VEL
LIN {X 0,Y 233.501,Z 780.921,A -85,B 0,C 180,E1 18952.56,E2 18952.56} C_VEL
LIN {X 0,Y 223.715,Z 802.272,A -85,B 0,C 180,E1 18960.612,E2 18960.612} C_VEL
LIN {X 0,Y 218.229,Z 818.223,A -85,B 0,C 180,E1 18969.699,E2 18969.699} C_VEL
LIN {X 0,Y 216.964,Z 827.34,A -85,B 0,C 180,E1 18977.912,E2 18977.912} C_VEL
LIN {X 0,Y 217.398,Z 831.954,A -85,B 0,C 180,E1 18986.003,E2 18986.003} C_VEL
LIN {X 0,Y 217.865,Z 832.65,A -85,B 0,C 180,E1 18989.996,E2 18989.996} C_VEL
LIN {X 0,Y 217.191,Z 830.245,A -85,B 0,C 180,E1 18998.01,E2 18998.01} C_VEL
LIN {X 0,Y 217.44,Z 822.21,A -85,B 0,C 180,E1 19007.209,E2 19007.209} C_VEL
LIN {X 0,Y 221.807,Z 807.346,A -85,B 0,C 180,E1 19016.919,E2 19016.919} C_VEL
LIN {X 0,Y 230.48,Z 787.37,A -85,B 0,C 180,E1 19025.376,E2 19025.376} C_VEL
LIN {X 0,Y 242.211,Z 762.818,A -85,B 0,C 180,E1 19032.3,E2 19032.3} C_VEL
LIN {X 0,Y 255.338,Z 733.521,A -85,B 0,C 180,E1 19037.828,E2 19037.828} C_VEL
LIN {X 0,Y 268.39,Z 700.067,A -85,B 0,C 180,E1 19041.899,E2 19041.899} C_VEL
LIN {X 0,Y 270.906,Z 690.61,A -85,B 0,C 180,E1 19042.908,E2 19042.908} C_VEL
LIN {X 0,Y 265.333,Z 667.809,A -85,B 0,C 180,E1 19047.818,E2 19047.818} C_VEL
LIN {X 0,Y 257.457,Z 647.417,A -85,B 0,C 180,E1 19053.288,E2 19053.288} C_VEL
LIN {X 0,Y 248.4,Z 629.16,A -85,B 0,C 180,E1 19059.781,E2 19059.781} C_VEL
LIN {X 0,Y 240.8,Z 616.616,A -85,B 0,C 180,E1 19066.489,E2 19066.489} C_VEL
LIN {X 0,Y 237.254,Z 610.56,A -85,B 0,C 180,E1 19070.83,E2 19070.83} C_VEL
LIN {X 0,Y 234.183,Z 604.366,A -85,B 0,C 180,E1 19077.115,E2 19077.115} C_VEL
LIN {X 0,Y 233.589,Z 604.243,A -85,B 0,C 180,E1 19088.06,E2 19088.06} C_VEL
LIN {X 0,Y 234.171,Z 607.839,A -85,B 0,C 180,E1 19091.011,E2 19091.011} C_VEL
LIN {X 0,Y 234.435,Z 613.281,A -85,B 0,C 180,E1 19093.552,E2 19093.552} C_VEL
LIN {X 0,Y 234.674,Z 619.661,A -85,B 0,C 180,E1 19096.032,E2 19096.032} C_VEL
LIN {X 0,Y 239.575,Z 630.153,A -85,B 0,C 180,E1 19103.276,E2 19103.276} C_VEL
LIN {X 0,Y 245.989,Z 647.38,A -85,B 0,C 180,E1 19111.231,E2 19111.231} C_VEL
LIN {X 0,Y 250.309,Z 663.868,A -85,B 0,C 180,E1 19117.231,E2 19117.231} C_VEL
LIN {X 0,Y 252.782,Z 683.074,A -85,B 0,C 180,E1 19123.372,E2 19123.372} C_VEL
LIN {X 0,Y 252.15,Z 700.611,A -85,B 0,C 180,E1 19128.667,E2 19128.667} C_VEL
LIN {X 0,Y 239.791,Z 723.274,A -85,B 0,C 180,E1 19134.269,E2 19134.269} C_VEL
LIN {X 0,Y 228.27,Z 741.873,A -85,B 0,C 180,E1 19141.262,E2 19141.262} C_VEL
LIN {X 0,Y 218.805,Z 755.831,A -85,B 0,C 180,E1 19149.763,E2 19149.763} C_VEL
LIN {X 0,Y 213.782,Z 763.39,A -85,B 0,C 180,E1 19157.737,E2 19157.737} C_VEL
LIN {X 0,Y 211.603,Z 766.972,A -85,B 0,C 180,E1 19165.901,E2 19165.901} C_VEL
LIN {X 0,Y 211.623,Z 766.936,A -85,B 0,C 180,E1 19174.106,E2 19174.106} C_VEL
LIN {X 0,Y 214.806,Z 761.793,A -85,B 0,C 180,E1 19184.286,E2 19184.286} C_VEL
LIN {X 0,Y 221.76,Z 751.419,A -85,B 0,C 180,E1 19193.296,E2 19193.296} C_VEL
LIN {X 0,Y 232.364,Z 735.324,A -85,B 0,C 180,E1 19201.421,E2 19201.421} C_VEL
LIN {X 0,Y 245.002,Z 714.036,A -85,B 0,C 180,E1 19208.172,E2 19208.172} C_VEL
LIN {X 0,Y 252.256,Z 699.109,A -85,B 0,C 180,E1 19211.653,E2 19211.653} C_VEL
LIN {X 0,Y 252.435,Z 680.055,A -85,B 0,C 180,E1 19217.443,E2 19217.443} C_VEL
LIN {X 0,Y 249.608,Z 660.995,A -85,B 0,C 180,E1 19223.575,E2 19223.575} C_VEL
LIN {X 0,Y 244.457,Z 643.258,A -85,B 0,C 180,E1 19230.288,E2 19230.288} C_VEL
LIN {X 0,Y 239.314,Z 629.873,A -85,B 0,C 180,E1 19236.698,E2 19236.698} C_VEL
LIN {X 0,Y 233.923,Z 618.091,A -85,B 0,C 180,E1 19244.985,E2 19244.985} C_VEL
LIN {X 0,Y 231.633,Z 612.257,A -85,B 0,C 180,E1 19251.664,E2 19251.664} C_VEL
LIN {X 0,Y 232.248,Z 611.566,A -85,B 0,C 180,E1 19262.325,E2 19262.325} C_VEL
LIN {X 0,Y 235.661,Z 618.334,A -85,B 0,C 180,E1 19269.504,E2 19269.504} C_VEL
LIN {X 0,Y 241.027,Z 628.639,A -85,B 0,C 180,E1 19275.976,E2 19275.976} C_VEL
LIN {X 0,Y 248.452,Z 642.457,A -85,B 0,C 180,E1 19282.362,E2 19282.362} C_VEL
LIN {X 0,Y 256.741,Z 662.286,A -85,B 0,C 180,E1 19288.758,E2 19288.758} C_VEL
LIN {X 0,Y 263.4,Z 686.012,A -85,B 0,C 180,E1 19294.573,E2 19294.573} C_VEL
LIN {X 0,Y 264.621,Z 694.954,A -85,B 0,C 180,E1 19296.401,E2 19296.401} C_VEL
LIN {X 0,Y 251.633,Z 728.162,A -85,B 0,C 180,E1 19300.232,E2 19300.232} C_VEL
LIN {X 0,Y 237.871,Z 757.857,A -85,B 0,C 180,E1 19305.557,E2 19305.557} C_VEL
LIN {X 0,Y 225.568,Z 782.499,A -85,B 0,C 180,E1 19312.227,E2 19312.227} C_VEL
LIN {X 0,Y 215.644,Z 803.14,A -85,B 0,C 180,E1 19320.559,E2 19320.559} C_VEL
LIN {X 0,Y 210.18,Z 818.588,A -85,B 0,C 180,E1 19330.21,E2 19330.21} C_VEL
LIN {X 0,Y 209.147,Z 827.71,A -85,B 0,C 180,E1 19339.615,E2 19339.615} C_VEL
LIN {X 0,Y 209.566,Z 830.761,A -85,B 0,C 180,E1 19345.853,E2 19345.853} C_VEL
LIN {X 0,Y 210.037,Z 831.461,A -85,B 0,C 180,E1 19349.996,E2 19349.996} C_VEL
LIN {X 0,Y 209.305,Z 829.035,A -85,B 0,C 180,E1 19358.314,E2 19358.314} C_VEL
LIN {X 0,Y 209.682,Z 821.036,A -85,B 0,C 180,E1 19367.808,E2 19367.808} C_VEL
LIN {X 0,Y 214.349,Z 806.416,A -85,B 0,C 180,E1 19377.738,E2 19377.738} C_VEL
LIN {X 0,Y 223.931,Z 785.89,A -85,B 0,C 180,E1 19386.67,E2 19386.67} C_VEL
LIN {X 0,Y 237.016,Z 759.913,A -85,B 0,C 180,E1 19393.997,E2 19393.997} C_VEL
LIN {X 0,Y 250.516,Z 730.971,A -85,B 0,C 180,E1 19399.391,E2 19399.391} C_VEL
LIN {X 0,Y 263.959,Z 697.205,A -85,B 0,C 180,E1 19403.414,E2 19403.414} C_VEL
LIN {X 0,Y 264.806,Z 693.35,A -85,B 0,C 180,E1 19403.899,E2 19403.899} C_VEL
LIN {X 0,Y 259.687,Z 671.035,A -85,B 0,C 180,E1 19409,E2 19409} C_VEL
LIN {X 0,Y 251.807,Z 649.779,A -85,B 0,C 180,E1 19415.12,E2 19415.12} C_VEL
LIN {X 0,Y 244.192,Z 634.272,A -85,B 0,C 180,E1 19421.262,E2 19421.262} C_VEL
LIN {X 0,Y 238.258,Z 623.698,A -85,B 0,C 180,E1 19427.16,E2 19427.16} C_VEL
LIN {X 0,Y 235.155,Z 617.93,A -85,B 0,C 180,E1 19431.448,E2 19431.448} C_VEL
LIN {X 0,Y 232.129,Z 611.516,A -85,B 0,C 180,E1 19438.843,E2 19438.843} C_VEL
LIN {X 0,Y 231.841,Z 612.474,A -85,B 0,C 180,E1 19448.122,E2 19448.122} C_VEL
LIN {X 0,Y 234.226,Z 618.227,A -85,B 0,C 180,E1 19454.995,E2 19454.995} C_VEL
LIN {X 0,Y 234.674,Z 619.661,A -85,B 0,C 180,E1 19456.032,E2 19456.032} C_VEL
LIN {X 0,Y 235.551,Z 628.56,A -85,B 0,C 180,E1 19459.711,E2 19459.711} C_VEL
LIN {X 0,Y 236.505,Z 638.087,A -85,B 0,C 180,E1 19463.321,E2 19463.321} C_VEL
LIN {X 0,Y 241.842,Z 654.491,A -85,B 0,C 180,E1 19471.108,E2 19471.108} C_VEL
LIN {X 0,Y 245.494,Z 671.979,A -85,B 0,C 180,E1 19477.616,E2 19477.616} C_VEL
LIN {X 0,Y 246.692,Z 690.166,A -85,B 0,C 180,E1 19483.626,E2 19483.626} C_VEL
LIN {X 0,Y 245.397,Z 703.616,A -85,B 0,C 180,E1 19487.834,E2 19487.834} C_VEL
LIN {X 0,Y 231.813,Z 727.247,A -85,B 0,C 180,E1 19494.003,E2 19494.003} C_VEL
LIN {X 0,Y 220.148,Z 744.897,A -85,B 0,C 180,E1 19501.227,E2 19501.227} C_VEL
LIN {X 0,Y 210.655,Z 758.247,A -85,B 0,C 180,E1 19510.042,E2 19510.042} C_VEL
LIN {X 0,Y 205.288,Z 765.832,A -85,B 0,C 180,E1 19519.379,E2 19519.379} C_VEL
LIN {X 0,Y 203.828,Z 768.156,A -85,B 0,C 180,E1 19525.744,E2 19525.744} C_VEL
LIN {X 0,Y 203.849,Z 768.12,A -85,B 0,C 180,E1 19534.263,E2 19534.263} C_VEL
LIN {X 0,Y 207.225,Z 762.986,A -85,B 0,C 180,E1 19544.82,E2 19544.82} C_VEL
LIN {X 0,Y 214.576,Z 752.64,A -85,B 0,C 180,E1 19554.103,E2 19554.103} C_VEL
LIN {X 0,Y 225.715,Z 736.539,A -85,B 0,C 180,E1 19562.458,E2 19562.458} C_VEL
LIN {X 0,Y 238.908,Z 715.27,A -85,B 0,C 180,E1 19569.33,E2 19569.33} C_VEL
LIN {X 0,Y 245.844,Z 701.5,A -85,B 0,C 180,E1 19572.647,E2 19572.647} C_VEL
LIN {X 0,Y 246.449,Z 682.887,A -85,B 0,C 180,E1 19578.574,E2 19578.574} C_VEL
LIN {X 0,Y 244.019,Z 663.769,A -85,B 0,C 180,E1 19585.121,E2 19585.121} C_VEL
LIN {X 0,Y 239.211,Z 646.075,A -85,B 0,C 180,E1 19592.393,E2 19592.393} C_VEL
LIN {X 0,Y 234.153,Z 631.951,A -85,B 0,C 180,E1 19600.145,E2 19600.145} C_VEL
LIN {X 0,Y 231.025,Z 625.046,A -85,B 0,C 180,E1 19606.15,E2 19606.15} C_VEL
LIN {X 0,Y 229.713,Z 619.292,A -85,B 0,C 180,E1 19612.415,E2 19612.415} C_VEL
LIN {X 0,Y 230.494,Z 619.631,A -85,B 0,C 180,E1 19622.578,E2 19622.578} C_VEL
LIN {X 0,Y 234.178,Z 627.723,A -85,B 0,C 180,E1 19630.368,E2 19630.368} C_VEL
LIN {X 0,Y 239.822,Z 638.358,A -85,B 0,C 180,E1 19637.068,E2 19637.068} C_VEL
LIN {X 0,Y 247.771,Z 656.117,A -85,B 0,C 180,E1 19644.348,E2 19644.348} C_VEL
LIN {X 0,Y 254.553,Z 676.209,A -85,B 0,C 180,E1 19650.358,E2 19650.358} C_VEL
LIN {X 0,Y 258.591,Z 695.637,A -85,B 0,C 180,E1 19655.036,E2 19655.036} C_VEL
LIN {X 0,Y 246.462,Z 726.776,A -85,B 0,C 180,E1 19658.79,E2 19658.79} C_VEL
LIN {X 0,Y 232.113,Z 756.547,A -85,B 0,C 180,E1 19664.146,E2 19664.146} C_VEL
LIN {X 0,Y 219.077,Z 781.334,A -85,B 0,C 180,E1 19670.952,E2 19670.952} C_VEL
LIN {X 0,Y 208.571,Z 801.884,A -85,B 0,C 180,E1 19679.456,E2 19679.456} C_VEL
LIN {X 0,Y 202.548,Z 817.254,A -85,B 0,C 180,E1 19689.353,E2 19689.353} C_VEL
LIN {X 0,Y 201.241,Z 825.624,A -85,B 0,C 180,E1 19697.915,E2 19697.915} C_VEL
LIN {X 0,Y 201.705,Z 829.563,A -85,B 0,C 180,E1 19705.691,E2 19705.691} C_VEL
LIN {X 0,Y 202.207,Z 830.272,A -85,B 0,C 180,E1 19709.996,E2 19709.996} C_VEL
LIN {X 0,Y 201.442,Z 827.828,A -85,B 0,C 180,E1 19718.641,E2 19718.641} C_VEL
LIN {X 0,Y 201.941,Z 819.876,A -85,B 0,C 180,E1 19728.439,E2 19728.439} C_VEL
LIN {X 0,Y 206.939,Z 805.467,A -85,B 0,C 180,E1 19738.628,E2 19738.628} C_VEL
LIN {X 0,Y 216.611,Z 786.047,A -85,B 0,C 180,E1 19747.432,E2 19747.432} C_VEL
LIN {X 0,Y 230.247,Z 760.466,A -85,B 0,C 180,E1 19754.977,E2 19754.977} C_VEL
LIN {X 0,Y 244.169,Z 732.026,A -85,B 0,C 180,E1 19760.458,E2 19760.458} C_VEL
LIN {X 0,Y 258.092,Z 698.891,A -85,B 0,C 180,E1 19764.546,E2 19764.546} C_VEL
LIN {X 0,Y 258.481,Z 694.369,A -85,B 0,C 180,E1 19765.293,E2 19765.293} C_VEL
LIN {X 0,Y 253.31,Z 671.468,A -85,B 0,C 180,E1 19770.957,E2 19770.957} C_VEL
LIN {X 0,Y 245.739,Z 651.079,A -85,B 0,C 180,E1 19777.534,E2 19777.534} C_VEL
LIN {X 0,Y 238.585,Z 636.328,A -85,B 0,C 180,E1 19784.301,E2 19784.301} C_VEL
LIN {X 0,Y 233.347,Z 625.711,A -85,B 0,C 180,E1 19791.322,E2 19791.322} C_VEL
LIN {X 0,Y 230.36,Z 619.21,A -85,B 0,C 180,E1 19798.775,E2 19798.775} C_VEL
LIN {X 0,Y 229.88,Z 620.08,A -85,B 0,C 180,E1 19807.818,E2 19807.818} C_VEL
LIN {X 0,Y 232.249,Z 627.752,A -85,B 0,C 180,E1 19816.095,E2 19816.095} C_VEL
LIN {X 0,Y 236.505,Z 638.087,A -85,B 0,C 180,E1 19823.321,E2 19823.321} C_VEL
LIN {X 0,Y 237.118,Z 642.785,A -85,B 0,C 180,E1 19825.108,E2 19825.108} C_VEL
LIN {X 0,Y 237.033,Z 659.496,A -85,B 0,C 180,E1 19830.107,E2 19830.107} C_VEL
LIN {X 0,Y 239.917,Z 676.283,A -85,B 0,C 180,E1 19836.729,E2 19836.729} C_VEL
LIN {X 0,Y 240.587,Z 693.741,A -85,B 0,C 180,E1 19842.796,E2 19842.796} C_VEL
LIN {X 0,Y 238.711,Z 706.622,A -85,B 0,C 180,E1 19846.959,E2 19846.959} C_VEL
LIN {X 0,Y 224.794,Z 729.549,A -85,B 0,C 180,E1 19853.215,E2 19853.215} C_VEL
LIN {X 0,Y 212.005,Z 747.921,A -85,B 0,C 180,E1 19861.185,E2 19861.185} C_VEL
LIN {X 0,Y 202.444,Z 760.503,A -85,B 0,C 180,E1 19870.338,E2 19870.338} C_VEL
LIN {X 0,Y 197.606,Z 767.019,A -85,B 0,C 180,E1 19878.961,E2 19878.961} C_VEL
LIN {X 0,Y 196.051,Z 769.341,A -85,B 0,C 180,E1 19885.575,E2 19885.575} C_VEL
LIN {X 0,Y 196.067,Z 769.306,A -85,B 0,C 180,E1 19894.433,E2 19894.433} C_VEL
LIN {X 0,Y 199.683,Z 764.175,A -85,B 0,C 180,E1 19905.393,E2 19905.393} C_VEL
LIN {X 0,Y 207.001,Z 754.464,A -85,B 0,C 180,E1 19914.532,E2 19914.532} C_VEL
LIN {X 0,Y 218.397,Z 738.887,A -85,B 0,C 180,E1 19923.092,E2 19923.092} C_VEL
LIN {X 0,Y 231.988,Z 718.026,A -85,B 0,C 180,E1 19930.13,E2 19930.13} C_VEL
LIN {X 0,Y 239.434,Z 704.416,A -85,B 0,C 180,E1 19933.495,E2 19933.495} C_VEL
LIN {X 0,Y 240.524,Z 686.114,A -85,B 0,C 180,E1 19939.647,E2 19939.647} C_VEL
LIN {X 0,Y 238.642,Z 667.437,A -85,B 0,C 180,E1 19946.411,E2 19946.411} C_VEL
LIN {X 0,Y 234.978,Z 651.968,A -85,B 0,C 180,E1 19953.179,E2 19953.179} C_VEL
LIN {X 0,Y 230.817,Z 638.656,A -85,B 0,C 180,E1 19960.843,E2 19960.843} C_VEL
LIN {X 0,Y 228.356,Z 632.296,A -85,B 0,C 180,E1 19966.571,E2 19966.571} C_VEL
LIN {X 0,Y 227.367,Z 626.798,A -85,B 0,C 180,E1 19973.297,E2 19973.297} C_VEL
LIN {X 0,Y 228.365,Z 627.415,A -85,B 0,C 180,E1 19982.405,E2 19982.405} C_VEL
LIN {X 0,Y 231.64,Z 635.24,A -85,B 0,C 180,E1 19990.076,E2 19990.076} C_VEL
LIN {X 0,Y 237.521,Z 647.558,A -85,B 0,C 180,E1 19997.613,E2 19997.613} C_VEL
LIN {X 0,Y 244.153,Z 663.687,A -85,B 0,C 180,E1 20004.246,E2 20004.246} C_VEL
LIN {X 0,Y 249.915,Z 683.485,A -85,B 0,C 180,E1 20010.243,E2 20010.243} C_VEL
LIN {X 0,Y 252.565,Z 699.551,A -85,B 0,C 180,E1 20014.198,E2 20014.198} C_VEL
LIN {X 0,Y 238.484,Z 731.613,A -85,B 0,C 180,E1 20018.216,E2 20018.216} C_VEL
LIN {X 0,Y 223.504,Z 760.815,A -85,B 0,C 180,E1 20023.962,E2 20023.962} C_VEL
LIN {X 0,Y 209.811,Z 785.266,A -85,B 0,C 180,E1 20031.435,E2 20031.435} C_VEL
LIN {X 0,Y 199.273,Z 805.183,A -85,B 0,C 180,E1 20040.839,E2 20040.839} C_VEL
LIN {X 0,Y 193.985,Z 819.591,A -85,B 0,C 180,E1 20051.804,E2 20051.804} C_VEL
LIN {X 0,Y 193.56,Z 826.595,A -85,B 0,C 180,E1 20060.996,E2 20060.996} C_VEL
LIN {X 0,Y 194.379,Z 829.083,A -85,B 0,C 180,E1 20069.996,E2 20069.996} C_VEL
LIN {X 0,Y 193.574,Z 826.619,A -85,B 0,C 180,E1 20078.995,E2 20078.995} C_VEL
LIN {X 0,Y 194.383,Z 818.118,A -85,B 0,C 180,E1 20089.706,E2 20089.706} C_VEL
LIN {X 0,Y 199.747,Z 804.203,A -85,B 0,C 180,E1 20099.76,E2 20099.76} C_VEL
LIN {X 0,Y 210.403,Z 784.357,A -85,B 0,C 180,E1 20108.951,E2 20108.951} C_VEL
LIN {X 0,Y 224.472,Z 759.144,A -85,B 0,C 180,E1 20116.469,E2 20116.469} C_VEL
LIN {X 0,Y 239.101,Z 730.681,A -85,B 0,C 180,E1 20121.952,E2 20121.952} C_VEL
LIN {X 0,Y 252.699,Z 699.597,A -85,B 0,C 180,E1 20125.823,E2 20125.823} C_VEL
LIN {X 0,Y 249.081,Z 679.428,A -85,B 0,C 180,E1 20130.915,E2 20130.915} C_VEL
LIN {X 0,Y 242.029,Z 657.858,A -85,B 0,C 180,E1 20137.966,E2 20137.966} C_VEL
LIN {X 0,Y 236.023,Z 644.122,A -85,B 0,C 180,E1 20144.285,E2 20144.285} C_VEL
LIN {X 0,Y 230.57,Z 632.809,A -85,B 0,C 180,E1 20152.153,E2 20152.153} C_VEL
LIN {X 0,Y 228.173,Z 626.732,A -85,B 0,C 180,E1 20159.387,E2 20159.387} C_VEL
LIN {X 0,Y 227.624,Z 627.658,A -85,B 0,C 180,E1 20167.535,E2 20167.535} C_VEL
LIN {X 0,Y 230.033,Z 636.882,A -85,B 0,C 180,E1 20177.239,E2 20177.239} C_VEL
LIN {X 0,Y 233.587,Z 647.178,A -85,B 0,C 180,E1 20184.1,E2 20184.1} C_VEL
LIN {X 0,Y 237.033,Z 659.496,A -85,B 0,C 180,E1 20190.107,E2 20190.107} C_VEL
LIN {X 0,Y 236.918,Z 667.585,A -85,B 0,C 180,E1 20192.602,E2 20192.602} C_VEL
LIN {X 0,Y 234.54,Z 682.579,A -85,B 0,C 180,E1 20196.563,E2 20196.563} C_VEL
LIN {X 0,Y 234.26,Z 699.589,A -85,B 0,C 180,E1 20202.752,E2 20202.752} C_VEL
LIN {X 0,Y 232.714,Z 708.545,A -85,B 0,C 180,E1 20205.803,E2 20205.803} C_VEL
LIN {X 0,Y 218.125,Z 731.413,A -85,B 0,C 180,E1 20212.22,E2 20212.22} C_VEL
LIN {X 0,Y 205.189,Z 749.119,A -85,B 0,C 180,E1 20220.133,E2 20220.133} C_VEL
LIN {X 0,Y 195.108,Z 761.69,A -85,B 0,C 180,E1 20229.566,E2 20229.566} C_VEL
LIN {X 0,Y 189.208,Z 769.242,A -85,B 0,C 180,E1 20240.795,E2 20240.795} C_VEL
LIN {X 0,Y 187.677,Z 771.044,A -85,B 0,C 180,E1 20250.004,E2 20250.004} C_VEL
LIN {X 0,Y 189.214,Z 769.188,A -85,B 0,C 180,E1 20259.213,E2 20259.213} C_VEL
LIN {X 0,Y 195.2,Z 761.541,A -85,B 0,C 180,E1 20270.432,E2 20270.432} C_VEL
LIN {X 0,Y 205.272,Z 748.87,A -85,B 0,C 180,E1 20279.863,E2 20279.863} C_VEL
LIN {X 0,Y 218.314,Z 731.008,A -85,B 0,C 180,E1 20287.78,E2 20287.78} C_VEL
LIN {X 0,Y 233.038,Z 707.415,A -85,B 0,C 180,E1 20294.37,E2 20294.37} C_VEL
LIN {X 0,Y 234.662,Z 689.447,A -85,B 0,C 180,E1 20300.741,E2 20300.741} C_VEL
LIN {X 0,Y 233.384,Z 671.789,A -85,B 0,C 180,E1 20307.501,E2 20307.501} C_VEL
LIN {X 0,Y 230.125,Z 655.711,A -85,B 0,C 180,E1 20315.074,E2 20315.074} C_VEL
LIN {X 0,Y 227.156,Z 644.757,A -85,B 0,C 180,E1 20322.078,E2 20322.078} C_VEL
LIN {X 0,Y 225.117,Z 638.708,A -85,B 0,C 180,E1 20328.349,E2 20328.349} C_VEL
LIN {X 0,Y 224.847,Z 635.358,A -85,B 0,C 180,E1 20332.25,E2 20332.25} C_VEL
LIN {X 0,Y 225.516,Z 634.071,A -85,B 0,C 180,E1 20339.989,E2 20339.989} C_VEL
LIN {X 0,Y 228.506,Z 641.18,A -85,B 0,C 180,E1 20348.867,E2 20348.867} C_VEL
LIN {X 0,Y 234.692,Z 655.703,A -85,B 0,C 180,E1 20357.833,E2 20357.833} C_VEL
LIN {X 0,Y 240.626,Z 672.607,A -85,B 0,C 180,E1 20364.625,E2 20364.625} C_VEL
LIN {X 0,Y 245.289,Z 692.255,A -85,B 0,C 180,E1 20370.572,E2 20370.572} C_VEL
LIN {X 0,Y 246.135,Z 702.875,A -85,B 0,C 180,E1 20373.152,E2 20373.152} C_VEL
LIN {X 0,Y 231.141,Z 735.06,A -85,B 0,C 180,E1 20377.414,E2 20377.414} C_VEL
LIN {X 0,Y 215.878,Z 762.969,A -85,B 0,C 180,E1 20383.306,E2 20383.306} C_VEL
LIN {X 0,Y 201.806,Z 786.736,A -85,B 0,C 180,E1 20391.068,E2 20391.068} C_VEL
LIN {X 0,Y 191.546,Z 805.085,A -85,B 0,C 180,E1 20400.371,E2 20400.371} C_VEL
LIN {X 0,Y 186.272,Z 818.352,A -85,B 0,C 180,E1 20411.023,E2 20411.023} C_VEL
LIN {X 0,Y 185.699,Z 825.384,A -85,B 0,C 180,E1 20420.611,E2 20420.611} C_VEL
LIN {X 0,Y 186.544,Z 827.893,A -85,B 0,C 180,E1 20429.996,E2 20429.996} C_VEL
LIN {X 0,Y 185.718,Z 825.41,A -85,B 0,C 180,E1 20439.379,E2 20439.379} C_VEL
LIN {X 0,Y 186.723,Z 816.875,A -85,B 0,C 180,E1 20450.55,E2 20450.55} C_VEL
LIN {X 0,Y 192.859,Z 802.563,A -85,B 0,C 180,E1 20461.196,E2 20461.196} C_VEL
LIN {X 0,Y 204.139,Z 782.948,A -85,B 0,C 180,E1 20470.458,E2 20470.458} C_VEL
LIN {X 0,Y 218.914,Z 757.837,A -85,B 0,C 180,E1 20478.023,E2 20478.023} C_VEL
LIN {X 0,Y 234.168,Z 729.33,A -85,B 0,C 180,E1 20483.522,E2 20483.522} C_VEL
LIN {X 0,Y 246.616,Z 701.081,A -85,B 0,C 180,E1 20487.185,E2 20487.185} C_VEL
LIN {X 0,Y 242.801,Z 679.79,A -85,B 0,C 180,E1 20493.059,E2 20493.059} C_VEL
LIN {X 0,Y 236.792,Z 660.929,A -85,B 0,C 180,E1 20499.91,E2 20499.91} C_VEL
LIN {X 0,Y 231.682,Z 648.755,A -85,B 0,C 180,E1 20506.187,E2 20506.187} C_VEL
LIN {X 0,Y 228.008,Z 640.232,A -85,B 0,C 180,E1 20512.379,E2 20512.379} C_VEL
LIN {X 0,Y 225.775,Z 634.192,A -85,B 0,C 180,E1 20520.011,E2 20520.011} C_VEL
LIN {X 0,Y 225.164,Z 634.171,A -85,B 0,C 180,E1 20523.866,E2 20523.866} C_VEL
LIN {X 0,Y 225.022,Z 637.568,A -85,B 0,C 180,E1 20529.695,E2 20529.695} C_VEL
LIN {X 0,Y 226.454,Z 642.325,A -85,B 0,C 180,E1 20535.523,E2 20535.523} C_VEL
LIN {X 0,Y 229.604,Z 653.283,A -85,B 0,C 180,E1 20543.318,E2 20543.318} C_VEL
LIN {X 0,Y 232.961,Z 668.252,A -85,B 0,C 180,E1 20550.813,E2 20550.813} C_VEL
LIN {X 0,Y 234.54,Z 682.579,A -85,B 0,C 180,E1 20556.563,E2 20556.563} C_VEL
LIN {X 0,Y 232.888,Z 691.091,A -85,B 0,C 180,E1 20558.982,E2 20558.982} C_VEL
LIN {X 0,Y 227.684,Z 705.889,A -85,B 0,C 180,E1 20562.914,E2 20562.914} C_VEL
LIN {X 0,Y 225.736,Z 712.211,A -85,B 0,C 180,E1 20564.999,E2 20564.999} C_VEL
LIN {X 0,Y 211.259,Z 733.65,A -85,B 0,C 180,E1 20571.301,E2 20571.301} C_VEL
LIN {X 0,Y 198.455,Z 750.316,A -85,B 0,C 180,E1 20579.01,E2 20579.01} C_VEL
LIN {X 0,Y 187.524,Z 763.184,A -85,B 0,C 180,E1 20589.055,E2 20589.055} C_VEL
LIN {X 0,Y 181.504,Z 770.427,A -85,B 0,C 180,E1 20600.401,E2 20600.401} C_VEL
LIN {X 0,Y 179.891,Z 772.227,A -85,B 0,C 180,E1 20610.004,E2 20610.004} C_VEL
LIN {X 0,Y 181.511,Z 770.374,A -85,B 0,C 180,E1 20619.608,E2 20619.608} C_VEL
LIN {X 0,Y 187.676,Z 762.963,A -85,B 0,C 180,E1 20631.021,E2 20631.021} C_VEL
LIN {X 0,Y 198.549,Z 750.069,A -85,B 0,C 180,E1 20640.983,E2 20640.983} C_VEL
LIN {X 0,Y 212.524,Z 731.795,A -85,B 0,C 180,E1 20649.221,E2 20649.221} C_VEL
LIN {X 0,Y 226.886,Z 709.518,A -85,B 0,C 180,E1 20655.61,E2 20655.61} C_VEL
LIN {X 0,Y 228.791,Z 692.343,A -85,B 0,C 180,E1 20662.032,E2 20662.032} C_VEL
LIN {X 0,Y 228.116,Z 675.216,A -85,B 0,C 180,E1 20669.032,E2 20669.032} C_VEL
LIN {X 0,Y 225.779,Z 660.908,A -85,B 0,C 180,E1 20676.263,E2 20676.263} C_VEL
LIN {X 0,Y 223.133,Z 649.766,A -85,B 0,C 180,E1 20684.24,E2 20684.24} C_VEL
LIN {X 0,Y 222.092,Z 643.072,A -85,B 0,C 180,E1 20692.153,E2 20692.153} C_VEL
LIN {X 0,Y 222.974,Z 641.58,A -85,B 0,C 180,E1 20699.989,E2 20699.989} C_VEL
LIN {X 0,Y 225.638,Z 648.703,A -85,B 0,C 180,E1 20708.673,E2 20708.673} C_VEL
LIN {X 0,Y 230.862,Z 662.05,A -85,B 0,C 180,E1 20717.154,E2 20717.154} C_VEL
LIN {X 0,Y 235.816,Z 677.858,A -85,B 0,C 180,E1 20723.786,E2 20723.786} C_VEL
LIN {X 0,Y 239.772,Z 696.881,A -85,B 0,C 180,E1 20729.807,E2 20729.807} C_VEL
LIN {X 0,Y 240.234,Z 705.094,A -85,B 0,C 180,E1 20731.932,E2 20731.932} C_VEL
LIN {X 0,Y 225.057,Z 735.978,A -85,B 0,C 180,E1 20736.164,E2 20736.164} C_VEL
LIN {X 0,Y 209.292,Z 763.371,A -85,B 0,C 180,E1 20742.136,E2 20742.136} C_VEL
LIN {X 0,Y 194.698,Z 786.759,A -85,B 0,C 180,E1 20750.088,E2 20750.088} C_VEL
LIN {X 0,Y 183.5,Z 805.586,A -85,B 0,C 180,E1 20760.322,E2 20760.322} C_VEL
LIN {X 0,Y 178.301,Z 818.25,A -85,B 0,C 180,E1 20771.427,E2 20771.427} C_VEL
LIN {X 0,Y 177.826,Z 824.171,A -85,B 0,C 180,E1 20780.191,E2 20780.191} C_VEL
LIN {X 0,Y 178.727,Z 826.705,A -85,B 0,C 180,E1 20789.996,E2 20789.996} C_VEL
LIN {X 0,Y 177.857,Z 824.2,A -85,B 0,C 180,E1 20799.798,E2 20799.798} C_VEL
LIN {X 0,Y 179.167,Z 815.411,A -85,B 0,C 180,E1 20811.673,E2 20811.673} C_VEL
LIN {X 0,Y 186.033,Z 801.08,A -85,B 0,C 180,E1 20822.642,E2 20822.642} C_VEL
LIN {X 0,Y 198.791,Z 780.352,A -85,B 0,C 180,E1 20832.521,E2 20832.521} C_VEL
LIN {X 0,Y 214.616,Z 754.676,A -85,B 0,C 180,E1 20840.096,E2 20840.096} C_VEL
LIN {X 0,Y 230.743,Z 725.57,A -85,B 0,C 180,E1 20845.51,E2 20845.51} C_VEL
LIN {X 0,Y 240.58,Z 703.454,A -85,B 0,C 180,E1 20848.427,E2 20848.427} C_VEL
LIN {X 0,Y 237.392,Z 683.503,A -85,B 0,C 180,E1 20854.313,E2 20854.313} C_VEL
LIN {X 0,Y 232.347,Z 666.149,A -85,B 0,C 180,E1 20860.996,E2 20860.996} C_VEL
LIN {X 0,Y 227.761,Z 654.246,A -85,B 0,C 180,E1 20867.534,E2 20867.534} C_VEL
LIN {X 0,Y 225.37,Z 647.918,A -85,B 0,C 180,E1 20872.289,E2 20872.289} C_VEL
LIN {X 0,Y 223.215,Z 641.759,A -85,B 0,C 180,E1 20880.011,E2 20880.011} C_VEL
LIN {X 0,Y 222.605,Z 641.708,A -85,B 0,C 180,E1 20883.911,E2 20883.911} C_VEL
LIN {X 0,Y 222.497,Z 646.459,A -85,B 0,C 180,E1 20891.79,E2 20891.79} C_VEL
LIN {X 0,Y 224.411,Z 654.286,A -85,B 0,C 180,E1 20899.185,E2 20899.185} C_VEL
LIN {X 0,Y 226.954,Z 666.896,A -85,B 0,C 180,E1 20906.775,E2 20906.775} C_VEL
LIN {X 0,Y 228.683,Z 681.235,A -85,B 0,C 180,E1 20913.371,E2 20913.371} C_VEL
LIN {X 0,Y 228.656,Z 698.234,A -85,B 0,C 180,E1 20920.069,E2 20920.069} C_VEL
LIN {X 0,Y 227.684,Z 705.889,A -85,B 0,C 180,E1 20922.914,E2 20922.914} C_VEL
LIN {X 0,Y 224.006,Z 711.853,A -85,B 0,C 180,E1 20924.194,E2 20924.194} C_VEL
LIN {X 0,Y 214.527,Z 722.105,A -85,B 0,C 180,E1 20925.82,E2 20925.82} C_VEL
LIN {X 0,Y 199.017,Z 742.843,A -85,B 0,C 180,E1 20933.234,E2 20933.234} C_VEL
LIN {X 0,Y 186.188,Z 757.82,A -85,B 0,C 180,E1 20942.128,E2 20942.128} C_VEL
LIN {X 0,Y 177.116,Z 767.869,A -85,B 0,C 180,E1 20952.596,E2 20952.596} C_VEL
LIN {X 0,Y 172.74,Z 772.893,A -85,B 0,C 180,E1 20964.976,E2 20964.976} C_VEL
LIN {X 0,Y 172.754,Z 772.86,A -85,B 0,C 180,E1 20975.033,E2 20975.033} C_VEL
LIN {X 0,Y 177.164,Z 767.749,A -85,B 0,C 180,E1 20987.409,E2 20987.409} C_VEL
LIN {X 0,Y 186.245,Z 757.633,A -85,B 0,C 180,E1 20997.872,E2 20997.872} C_VEL
LIN {X 0,Y 200.02,Z 741.387,A -85,B 0,C 180,E1 21007.273,E2 21007.273} C_VEL
LIN {X 0,Y 215.673,Z 720.194,A -85,B 0,C 180,E1 21014.593,E2 21014.593} C_VEL
LIN {X 0,Y 220.674,Z 712.307,A -85,B 0,C 180,E1 21016.663,E2 21016.663} C_VEL
LIN {X 0,Y 223.026,Z 695.256,A -85,B 0,C 180,E1 21023.39,E2 21023.39} C_VEL
LIN {X 0,Y 222.91,Z 679.404,A -85,B 0,C 180,E1 21030.304,E2 21030.304} C_VEL
LIN {X 0,Y 221.193,Z 665.551,A -85,B 0,C 180,E1 21037.873,E2 21037.873} C_VEL
LIN {X 0,Y 219.56,Z 655.359,A -85,B 0,C 180,E1 21045.819,E2 21045.819} C_VEL
LIN {X 0,Y 219.105,Z 650.67,A -85,B 0,C 180,E1 21052.053,E2 21052.053} C_VEL
LIN {X 0,Y 219.461,Z 649.001,A -85,B 0,C 180,E1 21056.033,E2 21056.033} C_VEL
LIN {X 0,Y 220.163,Z 649.012,A -85,B 0,C 180,E1 21059.989,E2 21059.989} C_VEL
LIN {X 0,Y 222.607,Z 656.558,A -85,B 0,C 180,E1 21068.792,E2 21068.792} C_VEL
LIN {X 0,Y 227.05,Z 668.959,A -85,B 0,C 180,E1 21076.832,E2 21076.832} C_VEL
LIN {X 0,Y 231.6,Z 685.953,A -85,B 0,C 180,E1 21084.001,E2 21084.001} C_VEL
LIN {X 0,Y 234.495,Z 705.044,A -85,B 0,C 180,E1 21090.1,E2 21090.1} C_VEL
LIN {X 0,Y 233.486,Z 709.261,A -85,B 0,C 180,E1 21090.894,E2 21090.894} C_VEL
LIN {X 0,Y 217.875,Z 739.052,A -85,B 0,C 180,E1 21095.257,E2 21095.257} C_VEL
LIN {X 0,Y 200.918,Z 766.592,A -85,B 0,C 180,E1 21101.687,E2 21101.687} C_VEL
LIN {X 0,Y 185.971,Z 789.09,A -85,B 0,C 180,E1 21110.143,E2 21110.143} C_VEL
LIN {X 0,Y 175.374,Z 806.264,A -85,B 0,C 180,E1 21120.397,E2 21120.397} C_VEL
LIN {X 0,Y 170.339,Z 818.088,A -85,B 0,C 180,E1 21131.87,E2 21131.87} C_VEL
LIN {X 0,Y 169.953,Z 822.956,A -85,B 0,C 180,E1 21139.732,E2 21139.732} C_VEL
LIN {X 0,Y 170.887,Z 825.514,A -85,B 0,C 180,E1 21149.995,E2 21149.995} C_VEL
LIN {X 0,Y 169.993,Z 822.987,A -85,B 0,C 180,E1 21160.256,E2 21160.256} C_VEL
LIN {X 0,Y 171.595,Z 814.165,A -85,B 0,C 180,E1 21172.682,E2 21172.682} C_VEL
LIN {X 0,Y 179.782,Z 798.886,A -85,B 0,C 180,E1 21184.636,E2 21184.636} C_VEL
LIN {X 0,Y 193.724,Z 777.647,A -85,B 0,C 180,E1 21194.693,E2 21194.693} C_VEL
LIN {X 0,Y 209.467,Z 753.375,A -85,B 0,C 180,E1 21201.811,E2 21201.811} C_VEL
LIN {X 0,Y 225.913,Z 724.868,A -85,B 0,C 180,E1 21207.106,E2 21207.106} C_VEL
LIN {X 0,Y 234.689,Z 706.411,A -85,B 0,C 180,E1 21209.573,E2 21209.573} C_VEL
LIN {X 0,Y 232.263,Z 688.46,A -85,B 0,C 180,E1 21215.148,E2 21215.148} C_VEL
LIN {X 0,Y 227.915,Z 671.449,A -85,B 0,C 180,E1 21222.073,E2 21222.073} C_VEL
LIN {X 0,Y 223.636,Z 659.343,A -85,B 0,C 180,E1 21229.281,E2 21229.281} C_VEL
LIN {X 0,Y 221.522,Z 653.978,A -85,B 0,C 180,E1 21234.127,E2 21234.127} C_VEL
LIN {X 0,Y 220.38,Z 649.232,A -85,B 0,C 180,E1 21240.011,E2 21240.011} C_VEL
LIN {X 0,Y 219.728,Z 649.125,A -85,B 0,C 180,E1 21243.962,E2 21243.962} C_VEL
LIN {X 0,Y 219.747,Z 655.711,A -85,B 0,C 180,E1 21254.169,E2 21254.169} C_VEL
LIN {X 0,Y 221.366,Z 665.881,A -85,B 0,C 180,E1 21262.108,E2 21262.108} C_VEL
LIN {X 0,Y 223.064,Z 679.863,A -85,B 0,C 180,E1 21269.74,E2 21269.74} C_VEL
LIN {X 0,Y 223.08,Z 696.913,A -85,B 0,C 180,E1 21277.137,E2 21277.137} C_VEL
LIN {X 0,Y 220.737,Z 712.615,A -85,B 0,C 180,E1 21283.321,E2 21283.321} C_VEL
LIN {X 0,Y 214.527,Z 722.105,A -85,B 0,C 180,E1 21285.82,E2 21285.82} C_VEL
LIN {X 0,Y 204.209,Z 733.008,A -85,B 0,C 180,E1 21288.332,E2 21288.332} C_VEL
LIN {X 0,Y 194.859,Z 741.635,A -85,B 0,C 180,E1 21290.79,E2 21290.79} C_VEL
LIN {X 0,Y 193.898,Z 742.749,A -85,B 0,C 180,E1 21291.261,E2 21291.261} C_VEL
LIN {X 0,Y 180.709,Z 757.581,A -85,B 0,C 180,E1 21299.827,E2 21299.827} C_VEL
LIN {X 0,Y 171.324,Z 767.3,A -85,B 0,C 180,E1 21309.304,E2 21309.304} C_VEL
LIN {X 0,Y 166.121,Z 772.798,A -85,B 0,C 180,E1 21319.502,E2 21319.502} C_VEL
LIN {X 0,Y 164.296,Z 774.596,A -85,B 0,C 180,E1 21330.005,E2 21330.005} C_VEL
LIN {X 0,Y 166.128,Z 772.746,A -85,B 0,C 180,E1 21340.507,E2 21340.507} C_VEL
LIN {X 0,Y 172.673,Z 765.853,A -85,B 0,C 180,E1 21352.296,E2 21352.296} C_VEL
LIN {X 0,Y 183.721,Z 754.173,A -85,B 0,C 180,E1 21362.393,E2 21362.393} C_VEL
LIN {X 0,Y 198.645,Z 736.749,A -85,B 0,C 180,E1 21371.105,E2 21371.105} C_VEL
LIN {X 0,Y 214.183,Z 715.57,A -85,B 0,C 180,E1 21377.603,E2 21377.603} C_VEL
LIN {X 0,Y 217.231,Z 700.024,A -85,B 0,C 180,E1 21384.038,E2 21384.038} C_VEL
LIN {X 0,Y 217.841,Z 685.06,A -85,B 0,C 180,E1 21390.876,E2 21390.876} C_VEL
LIN {X 0,Y 216.909,Z 671.411,A -85,B 0,C 180,E1 21398.714,E2 21398.714} C_VEL
LIN {X 0,Y 215.983,Z 662.912,A -85,B 0,C 180,E1 21405.579,E2 21405.579} C_VEL
LIN {X 0,Y 215.828,Z 658.095,A -85,B 0,C 180,E1 21412.054,E2 21412.054} C_VEL
LIN {X 0,Y 216.349,Z 656.342,A -85,B 0,C 180,E1 21415.976,E2 21415.976} C_VEL
LIN {X 0,Y 217.122,Z 656.388,A -85,B 0,C 180,E1 21419.989,E2 21419.989} C_VEL
LIN {X 0,Y 219.771,Z 665.572,A -85,B 0,C 180,E1 21430.03,E2 21430.03} C_VEL
LIN {X 0,Y 223.795,Z 678.578,A -85,B 0,C 180,E1 21437.916,E2 21437.916} C_VEL
LIN {X 0,Y 227.499,Z 696.615,A -85,B 0,C 180,E1 21445.228,E2 21445.228} C_VEL
LIN {X 0,Y 228.666,Z 709.175,A -85,B 0,C 180,E1 21449.272,E2 21449.272} C_VEL
LIN {X 0,Y 211.999,Z 739.918,A -85,B 0,C 180,E1 21453.873,E2 21453.873} C_VEL
LIN {X 0,Y 194.176,Z 767.285,A -85,B 0,C 180,E1 21460.506,E2 21460.506} C_VEL
LIN {X 0,Y 178.765,Z 789.219,A -85,B 0,C 180,E1 21469.14,E2 21469.14} C_VEL
LIN {X 0,Y 167.265,Z 806.729,A -85,B 0,C 180,E1 21480.434,E2 21480.434} C_VEL
LIN {X 0,Y 162.623,Z 816.85,A -85,B 0,C 180,E1 21490.978,E2 21490.978} C_VEL
LIN {X 0,Y 162.058,Z 821.736,A -85,B 0,C 180,E1 21499.226,E2 21499.226} C_VEL
LIN {X 0,Y 163.072,Z 824.327,A -85,B 0,C 180,E1 21509.995,E2 21509.995} C_VEL
LIN {X 0,Y 162.102,Z 821.768,A -85,B 0,C 180,E1 21520.761,E2 21520.761} C_VEL
LIN {X 0,Y 163.79,Z 813.611,A -85,B 0,C 180,E1 21533.035,E2 21533.035} C_VEL
LIN {X 0,Y 171.777,Z 799.56,A -85,B 0,C 180,E1 21544.947,E2 21544.947} C_VEL
LIN {X 0,Y 186.027,Z 779.126,A -85,B 0,C 180,E1 21555.403,E2 21555.403} C_VEL
LIN {X 0,Y 203.557,Z 753.536,A -85,B 0,C 180,E1 21563.267,E2 21563.267} C_VEL
LIN {X 0,Y 220.493,Z 725.492,A -85,B 0,C 180,E1 21568.572,E2 21568.572} C_VEL
LIN {X 0,Y 228.813,Z 709.364,A -85,B 0,C 180,E1 21570.711,E2 21570.711} C_VEL
LIN {X 0,Y 226.612,Z 691.043,A -85,B 0,C 180,E1 21576.9,E2 21576.9} C_VEL
LIN {X 0,Y 223.047,Z 675.612,A -85,B 0,C 180,E1 21583.7,E2 21583.7} C_VEL
LIN {X 0,Y 219.137,Z 663.192,A -85,B 0,C 180,E1 21592.069,E2 21592.069} C_VEL
LIN {X 0,Y 217.314,Z 656.639,A -85,B 0,C 180,E1 21600.011,E2 21600.011} C_VEL
LIN {X 0,Y 216.598,Z 656.492,A -85,B 0,C 180,E1 21604.019,E2 21604.019} C_VEL
LIN {X 0,Y 216.156,Z 663.251,A -85,B 0,C 180,E1 21614.409,E2 21614.409} C_VEL
LIN {X 0,Y 217.239,Z 673.231,A -85,B 0,C 180,E1 21622.286,E2 21622.286} C_VEL
LIN {X 0,Y 218.015,Z 686.789,A -85,B 0,C 180,E1 21629.799,E2 21629.799} C_VEL
LIN {X 0,Y 216.961,Z 703.4,A -85,B 0,C 180,E1 21637.285,E2 21637.285} C_VEL
LIN {X 0,Y 214.173,Z 715.857,A -85,B 0,C 180,E1 21642.341,E2 21642.341} C_VEL
LIN {X 0,Y 197.581,Z 738.322,A -85,B 0,C 180,E1 21649.363,E2 21649.363} C_VEL
LIN {X 0,Y 193.898,Z 742.749,A -85,B 0,C 180,E1 21651.261,E2 21651.261} C_VEL
LIN {X 0,Y 183.804,Z 751.526,A -85,B 0,C 180,E1 21654.702,E2 21654.702} C_VEL
LIN {X 0,Y 173.819,Z 758.943,A -85,B 0,C 180,E1 21658.674,E2 21658.674} C_VEL
LIN {X 0,Y 164.044,Z 768.486,A -85,B 0,C 180,E1 21668.341,E2 21668.341} C_VEL
LIN {X 0,Y 158.446,Z 773.984,A -85,B 0,C 180,E1 21678.988,E2 21678.988} C_VEL
LIN {X 0,Y 156.487,Z 775.783,A -85,B 0,C 180,E1 21690.005,E2 21690.005} C_VEL
LIN {X 0,Y 158.454,Z 773.933,A -85,B 0,C 180,E1 21701.022,E2 21701.022} C_VEL
LIN {X 0,Y 165.712,Z 766.803,A -85,B 0,C 180,E1 21713.608,E2 21713.608} C_VEL
LIN {X 0,Y 178.827,Z 753.676,A -85,B 0,C 180,E1 21724.859,E2 21724.859} C_VEL
LIN {X 0,Y 194.946,Z 735.434,A -85,B 0,C 180,E1 21733.578,E2 21733.578} C_VEL
LIN {X 0,Y 208.478,Z 717.255,A -85,B 0,C 180,E1 21739.171,E2 21739.171} C_VEL
LIN {X 0,Y 211.787,Z 701.832,A -85,B 0,C 180,E1 21745.984,E2 21745.984} C_VEL
LIN {X 0,Y 212.73,Z 687.769,A -85,B 0,C 180,E1 21753.005,E2 21753.005} C_VEL
LIN {X 0,Y 212.421,Z 674.997,A -85,B 0,C 180,E1 21761.183,E2 21761.183} C_VEL
LIN {X 0,Y 212.098,Z 667.236,A -85,B 0,C 180,E1 21769.221,E2 21769.221} C_VEL
LIN {X 0,Y 213.007,Z 663.616,A -85,B 0,C 180,E1 21775.913,E2 21775.913} C_VEL
LIN {X 0,Y 213.864,Z 663.671,A -85,B 0,C 180,E1 21779.989,E2 21779.989} C_VEL
LIN {X 0,Y 215.821,Z 671.733,A -85,B 0,C 180,E1 21789.133,E2 21789.133} C_VEL
LIN {X 0,Y 219.235,Z 684.332,A -85,B 0,C 180,E1 21797.16,E2 21797.16} C_VEL
LIN {X 0,Y 222.049,Z 700.666,A -85,B 0,C 180,E1 21804.137,E2 21804.137} C_VEL
LIN {X 0,Y 222.262,Z 713.054,A -85,B 0,C 180,E1 21808.128,E2 21808.128} C_VEL
LIN {X 0,Y 204.276,Z 743.725,A -85,B 0,C 180,E1 21813.017,E2 21813.017} C_VEL
LIN {X 0,Y 185.584,Z 770.646,A -85,B 0,C 180,E1 21820.105,E2 21820.105} C_VEL
LIN {X 0,Y 169.548,Z 792.099,A -85,B 0,C 180,E1 21829.615,E2 21829.615} C_VEL
LIN {X 0,Y 158.485,Z 808.225,A -85,B 0,C 180,E1 21841.462,E2 21841.462} C_VEL
LIN {X 0,Y 154.421,Z 817.509,A -85,B 0,C 180,E1 21852.889,E2 21852.889} C_VEL
LIN {X 0,Y 154.472,Z 822.359,A -85,B 0,C 180,E1 21864.37,E2 21864.37} C_VEL
LIN {X 0,Y 155.224,Z 823.135,A -85,B 0,C 180,E1 21869.995,E2 21869.995} C_VEL
LIN {X 0,Y 154.213,Z 820.548,A -85,B 0,C 180,E1 21881.319,E2 21881.319} C_VEL
LIN {X 0,Y 156.331,Z 812.294,A -85,B 0,C 180,E1 21894.3,E2 21894.3} C_VEL
LIN {X 0,Y 165.096,Z 798.299,A -85,B 0,C 180,E1 21906.584,E2 21906.584} C_VEL
LIN {X 0,Y 179.345,Z 779.158,A -85,B 0,C 180,E1 21916.722,E2 21916.722} C_VEL
LIN {X 0,Y 197.443,Z 754.22,A -85,B 0,C 180,E1 21924.684,E2 21924.684} C_VEL
LIN {X 0,Y 215.293,Z 725.988,A -85,B 0,C 180,E1 21930.13,E2 21930.13} C_VEL
LIN {X 0,Y 222.918,Z 711.508,A -85,B 0,C 180,E1 21932.195,E2 21932.195} C_VEL
LIN {X 0,Y 221.222,Z 694.339,A -85,B 0,C 180,E1 21938.428,E2 21938.428} C_VEL
LIN {X 0,Y 218.418,Z 680.487,A -85,B 0,C 180,E1 21945.048,E2 21945.048} C_VEL
LIN {X 0,Y 215.64,Z 670.679,A -85,B 0,C 180,E1 21951.939,E2 21951.939} C_VEL
LIN {X 0,Y 214.032,Z 663.946,A -85,B 0,C 180,E1 21960.011,E2 21960.011} C_VEL
LIN {X 0,Y 212.893,Z 664.379,A -85,B 0,C 180,E1 21965.398,E2 21965.398} C_VEL
LIN {X 0,Y 212.386,Z 671.478,A -85,B 0,C 180,E1 21975.517,E2 21975.517} C_VEL
LIN {X 0,Y 212.809,Z 681.401,A -85,B 0,C 180,E1 21983.045,E2 21983.045} C_VEL
LIN {X 0,Y 212.562,Z 694.981,A -85,B 0,C 180,E1 21990.556,E2 21990.556} C_VEL
LIN {X 0,Y 210.238,Z 711.274,A -85,B 0,C 180,E1 21998.109,E2 21998.109} C_VEL
LIN {X 0,Y 207.362,Z 719.446,A -85,B 0,C 180,E1 22001.355,E2 22001.355} C_VEL
LIN {X 0,Y 190.695,Z 740.676,A -85,B 0,C 180,E1 22008.329,E2 22008.329} C_VEL
LIN {X 0,Y 175.517,Z 757.203,A -85,B 0,C 180,E1 22017.381,E2 22017.381} C_VEL
LIN {X 0,Y 173.819,Z 758.943,A -85,B 0,C 180,E1 22018.674,E2 22018.674} C_VEL
LIN {X 0,Y 164.437,Z 765.302,A -85,B 0,C 180,E1 22023.232,E2 22023.232} C_VEL
LIN {X 0,Y 155.974,Z 770.405,A -85,B 0,C 180,E1 22028.409,E2 22028.409} C_VEL
LIN {X 0,Y 150.785,Z 775.17,A -85,B 0,C 180,E1 22038.421,E2 22038.421} C_VEL
LIN {X 0,Y 148.677,Z 776.969,A -85,B 0,C 180,E1 22050.005,E2 22050.005} C_VEL
LIN {X 0,Y 150.794,Z 775.119,A -85,B 0,C 180,E1 22061.59,E2 22061.59} C_VEL
LIN {X 0,Y 158.164,Z 768.377,A -85,B 0,C 180,E1 22074.265,E2 22074.265} C_VEL
LIN {X 0,Y 170.706,Z 756.566,A -85,B 0,C 180,E1 22085.21,E2 22085.21} C_VEL
LIN {X 0,Y 187.156,Z 739.181,A -85,B 0,C 180,E1 22094.251,E2 22094.251} C_VEL
LIN {X 0,Y 202.267,Z 720.36,A -85,B 0,C 180,E1 22100.287,E2 22100.287} C_VEL
LIN {X 0,Y 206.149,Z 705.403,A -85,B 0,C 180,E1 22107.225,E2 22107.225} C_VEL
LIN {X 0,Y 207.615,Z 692.581,A -85,B 0,C 180,E1 22114.039,E2 22114.039} C_VEL
LIN {X 0,Y 208.064,Z 680.949,A -85,B 0,C 180,E1 22121.973,E2 22121.973} C_VEL
LIN {X 0,Y 208.27,Z 674.036,A -85,B 0,C 180,E1 22129.517,E2 22129.517} C_VEL
LIN {X 0,Y 209.448,Z 670.771,A -85,B 0,C 180,E1 22135.843,E2 22135.843} C_VEL
LIN {X 0,Y 210.298,Z 670.835,A -85,B 0,C 180,E1 22139.988,E2 22139.988} C_VEL
LIN {X 0,Y 212.091,Z 679.078,A -85,B 0,C 180,E1 22149.295,E2 22149.295} C_VEL
LIN {X 0,Y 214.76,Z 690.984,A -85,B 0,C 180,E1 22156.894,E2 22156.894} C_VEL
LIN {X 0,Y 216.73,Z 707.648,A -85,B 0,C 180,E1 22164.138,E2 22164.138} C_VEL
LIN {X 0,Y 216.699,Z 715.044,A -85,B 0,C 180,E1 22166.682,E2 22166.682} C_VEL
LIN {X 0,Y 198.594,Z 744.421,A -85,B 0,C 180,E1 22171.464,E2 22171.464} C_VEL
LIN {X 0,Y 179.261,Z 770.785,A -85,B 0,C 180,E1 22178.618,E2 22178.618} C_VEL
LIN {X 0,Y 163.067,Z 791.187,A -85,B 0,C 180,E1 22187.946,E2 22187.946} C_VEL
LIN {X 0,Y 151.329,Z 806.971,A -85,B 0,C 180,E1 22199.978,E2 22199.978} C_VEL
LIN {X 0,Y 146.684,Z 816.274,A -85,B 0,C 180,E1 22211.956,E2 22211.956} C_VEL
LIN {X 0,Y 146.582,Z 821.155,A -85,B 0,C 180,E1 22224.066,E2 22224.066} C_VEL
LIN {X 0,Y 147.385,Z 821.944,A -85,B 0,C 180,E1 22229.995,E2 22229.995} C_VEL
LIN {X 0,Y 146.355,Z 819.329,A -85,B 0,C 180,E1 22241.935,E2 22241.935} C_VEL
LIN {X 0,Y 148.938,Z 811.055,A -85,B 0,C 180,E1 22255.591,E2 22255.591} C_VEL
LIN {X 0,Y 158.555,Z 797.037,A -85,B 0,C 180,E1 22268.359,E2 22268.359} C_VEL
LIN {X 0,Y 173.826,Z 777.892,A -85,B 0,C 180,E1 22278.691,E2 22278.691} C_VEL
LIN {X 0,Y 192.904,Z 752.82,A -85,B 0,C 180,E1 22286.689,E2 22286.689} C_VEL
LIN {X 0,Y 210.905,Z 725.416,A -85,B 0,C 180,E1 22291.922,E2 22291.922} C_VEL
LIN {X 0,Y 216.755,Z 715.345,A -85,B 0,C 180,E1 22293.293,E2 22293.293} C_VEL
LIN {X 0,Y 216.29,Z 701.176,A -85,B 0,C 180,E1 22298.53,E2 22298.53} C_VEL
LIN {X 0,Y 213.969,Z 686.549,A -85,B 0,C 180,E1 22305.673,E2 22305.673} C_VEL
LIN {X 0,Y 211.36,Z 675.968,A -85,B 0,C 180,E1 22313.843,E2 22313.843} C_VEL
LIN {X 0,Y 210.456,Z 671.129,A -85,B 0,C 180,E1 22320.011,E2 22320.011} C_VEL
LIN {X 0,Y 209.274,Z 671.532,A -85,B 0,C 180,E1 22325.492,E2 22325.492} C_VEL
LIN {X 0,Y 208.269,Z 678.141,A -85,B 0,C 180,E1 22335.189,E2 22335.189} C_VEL
LIN {X 0,Y 207.995,Z 687.987,A -85,B 0,C 180,E1 22342.886,E2 22342.886} C_VEL
LIN {X 0,Y 206.917,Z 700.968,A -85,B 0,C 180,E1 22350.331,E2 22350.331} C_VEL
LIN {X 0,Y 204.138,Z 715.214,A -85,B 0,C 180,E1 22357.246,E2 22357.246} C_VEL
LIN {X 0,Y 202.249,Z 720.694,A -85,B 0,C 180,E1 22359.681,E2 22359.681} C_VEL
LIN {X 0,Y 184.935,Z 741.878,A -85,B 0,C 180,E1 22366.72,E2 22366.72} C_VEL
LIN {X 0,Y 168.996,Z 758.396,A -85,B 0,C 180,E1 22375.955,E2 22375.955} C_VEL
LIN {X 0,Y 156.818,Z 769.67,A -85,B 0,C 180,E1 22387.288,E2 22387.288} C_VEL
LIN {X 0,Y 155.974,Z 770.405,A -85,B 0,C 180,E1 22388.409,E2 22388.409} C_VEL
LIN {X 0,Y 148.524,Z 774.357,A -85,B 0,C 180,E1 22394.197,E2 22394.197} C_VEL
LIN {X 0,Y 142.262,Z 776.947,A -85,B 0,C 180,E1 22400.589,E2 22400.589} C_VEL
LIN {X 0,Y 140.868,Z 778.155,A -85,B 0,C 180,E1 22410.006,E2 22410.006} C_VEL
LIN {X 0,Y 143.148,Z 776.306,A -85,B 0,C 180,E1 22422.218,E2 22422.218} C_VEL
LIN {X 0,Y 151.183,Z 769.458,A -85,B 0,C 180,E1 22435.633,E2 22435.633} C_VEL
LIN {X 0,Y 164.378,Z 757.763,A -85,B 0,C 180,E1 22446.782,E2 22446.782} C_VEL
LIN {X 0,Y 181.656,Z 740.392,A -85,B 0,C 180,E1 22455.966,E2 22455.966} C_VEL
LIN {X 0,Y 196.733,Z 722.202,A -85,B 0,C 180,E1 22461.984,E2 22461.984} C_VEL
LIN {X 0,Y 200.801,Z 707.783,A -85,B 0,C 180,E1 22469.195,E2 22469.195} C_VEL
LIN {X 0,Y 202.645,Z 696.149,A -85,B 0,C 180,E1 22475.937,E2 22475.937} C_VEL
LIN {X 0,Y 203.706,Z 685.726,A -85,B 0,C 180,E1 22483.805,E2 22483.805} C_VEL
LIN {X 0,Y 204.632,Z 679.463,A -85,B 0,C 180,E1 22492.145,E2 22492.145} C_VEL
LIN {X 0,Y 205.562,Z 677.809,A -85,B 0,C 180,E1 22495.764,E2 22495.764} C_VEL
LIN {X 0,Y 206.495,Z 677.882,A -85,B 0,C 180,E1 22499.988,E2 22499.988} C_VEL
LIN {X 0,Y 208.074,Z 686.288,A -85,B 0,C 180,E1 22509.411,E2 22509.411} C_VEL
LIN {X 0,Y 210.041,Z 697.732,A -85,B 0,C 180,E1 22516.746,E2 22516.746} C_VEL
LIN {X 0,Y 211.158,Z 712.865,A -85,B 0,C 180,E1 22523.527,E2 22523.527} C_VEL
LIN {X 0,Y 211.031,Z 717.391,A -85,B 0,C 180,E1 22525.209,E2 22525.209} C_VEL
LIN {X 0,Y 192.377,Z 746.092,A -85,B 0,C 180,E1 22530.028,E2 22530.028} C_VEL
LIN {X 0,Y 173.07,Z 770.931,A -85,B 0,C 180,E1 22537.028,E2 22537.028} C_VEL
LIN {X 0,Y 155.535,Z 791.755,A -85,B 0,C 180,E1 22547.04,E2 22547.04} C_VEL
LIN {X 0,Y 143.27,Z 807.091,A -85,B 0,C 180,E1 22559.864,E2 22559.864} C_VEL
LIN {X 0,Y 138.526,Z 816.663,A -85,B 0,C 180,E1 22574.137,E2 22574.137} C_VEL
LIN {X 0,Y 138.688,Z 819.948,A -85,B 0,C 180,E1 22583.727,E2 22583.727} C_VEL
LIN {X 0,Y 139.527,Z 820.75,A -85,B 0,C 180,E1 22589.994,E2 22589.994} C_VEL
LIN {X 0,Y 138.472,Z 818.104,A -85,B 0,C 180,E1 22602.625,E2 22602.625} C_VEL
LIN {X 0,Y 141.599,Z 809.811,A -85,B 0,C 180,E1 22617.021,E2 22617.021} C_VEL
LIN {X 0,Y 152.206,Z 795.783,A -85,B 0,C 180,E1 22630.276,E2 22630.276} C_VEL
LIN {X 0,Y 169.357,Z 775.718,A -85,B 0,C 180,E1 22641.156,E2 22641.156} C_VEL
LIN {X 0,Y 189.273,Z 750.465,A -85,B 0,C 180,E1 22649.025,E2 22649.025} C_VEL
LIN {X 0,Y 208.366,Z 722.235,A -85,B 0,C 180,E1 22654.166,E2 22654.166} C_VEL
LIN {X 0,Y 211.29,Z 716.538,A -85,B 0,C 180,E1 22655.116,E2 22655.116} C_VEL
LIN {X 0,Y 210.469,Z 700.057,A -85,B 0,C 180,E1 22662.157,E2 22662.157} C_VEL
LIN {X 0,Y 208.452,Z 687.869,A -85,B 0,C 180,E1 22669.55,E2 22669.55} C_VEL
LIN {X 0,Y 206.687,Z 679.696,A -85,B 0,C 180,E1 22677.913,E2 22677.913} C_VEL
LIN {X 0,Y 206.63,Z 678.181,A -85,B 0,C 180,E1 22680.012,E2 22680.012} C_VEL
LIN {X 0,Y 205.794,Z 677.955,A -85,B 0,C 180,E1 22684.231,E2 22684.231} C_VEL
LIN {X 0,Y 204.058,Z 683.943,A -85,B 0,C 180,E1 22694.029,E2 22694.029} C_VEL
LIN {X 0,Y 203.131,Z 693.192,A -85,B 0,C 180,E1 22701.893,E2 22701.893} C_VEL
LIN {X 0,Y 201.558,Z 704.778,A -85,B 0,C 180,E1 22708.976,E2 22708.976} C_VEL
LIN {X 0,Y 197.849,Z 719.487,A -85,B 0,C 180,E1 22716.568,E2 22716.568} C_VEL
LIN {X 0,Y 195.57,Z 724.268,A -85,B 0,C 180,E1 22718.574,E2 22718.574} C_VEL
LIN {X 0,Y 177.151,Z 745.365,A -85,B 0,C 180,E1 22726.027,E2 22726.027} C_VEL
LIN {X 0,Y 160.878,Z 761.149,A -85,B 0,C 180,E1 22735.627,E2 22735.627} C_VEL
LIN {X 0,Y 148.572,Z 771.732,A -85,B 0,C 180,E1 22747.526,E2 22747.526} C_VEL
LIN {X 0,Y 142.262,Z 776.947,A -85,B 0,C 180,E1 22760.589,E2 22760.589} C_VEL
LIN {X 0,Y 138.74,Z 778.317,A -85,B 0,C 180,E1 22765.714,E2 22765.714} C_VEL
LIN {X 0,Y 133.446,Z 779.121,A -85,B 0,C 180,E1 22774.232,E2 22774.232} C_VEL
LIN {X 0,Y 133.507,Z 778.943,A -85,B 0,C 180,E1 22774.703,E2 22774.703} C_VEL
LIN {X 0,Y 138.371,Z 775.183,A -85,B 0,C 180,E1 22789.169,E2 22789.169} C_VEL
LIN {X 0,Y 149.55,Z 766.333,A -85,B 0,C 180,E1 22802.113,E2 22802.113} C_VEL
LIN {X 0,Y 165.489,Z 752.335,A -85,B 0,C 180,E1 22812.705,E2 22812.705} C_VEL
LIN {X 0,Y 183.603,Z 733.708,A -85,B 0,C 180,E1 22820.638,E2 22820.638} C_VEL
LIN {X 0,Y 190.856,Z 724.959,A -85,B 0,C 180,E1 22823.391,E2 22823.391} C_VEL
LIN {X 0,Y 195.45,Z 711.165,A -85,B 0,C 180,E1 22830.722,E2 22830.722} C_VEL
LIN {X 0,Y 197.928,Z 699.24,A -85,B 0,C 180,E1 22838.296,E2 22838.296} C_VEL
LIN {X 0,Y 199.374,Z 690.598,A -85,B 0,C 180,E1 22845.7,E2 22845.7} C_VEL
LIN {X 0,Y 200.469,Z 686.287,A -85,B 0,C 180,E1 22852.204,E2 22852.204} C_VEL
LIN {X 0,Y 201.465,Z 684.718,A -85,B 0,C 180,E1 22855.678,E2 22855.678} C_VEL
LIN {X 0,Y 202.49,Z 684.802,A -85,B 0,C 180,E1 22859.988,E2 22859.988} C_VEL
LIN {X 0,Y 203.718,Z 693.174,A -85,B 0,C 180,E1 22869.418,E2 22869.418} C_VEL
LIN {X 0,Y 205.035,Z 703.637,A -85,B 0,C 180,E1 22876.257,E2 22876.257} C_VEL
LIN {X 0,Y 205.447,Z 718.917,A -85,B 0,C 180,E1 22883.292,E2 22883.292} C_VEL
LIN {X 0,Y 201.963,Z 725.242,A -85,B 0,C 180,E1 22884.437,E2 22884.437} C_VEL
LIN {X 0,Y 181.494,Z 753.858,A -85,B 0,C 180,E1 22890.019,E2 22890.019} C_VEL
LIN {X 0,Y 162.467,Z 776.294,A -85,B 0,C 180,E1 22897.438,E2 22897.438} C_VEL
LIN {X 0,Y 145.741,Z 794.705,A -85,B 0,C 180,E1 22907.829,E2 22907.829} C_VEL
LIN {X 0,Y 134.324,Z 808.5,A -85,B 0,C 180,E1 22921.371,E2 22921.371} C_VEL
LIN {X 0,Y 130.579,Z 816.847,A -85,B 0,C 180,E1 22936.585,E2 22936.585} C_VEL
LIN {X 0,Y 131.694,Z 819.56,A -85,B 0,C 180,E1 22949.994,E2 22949.994} C_VEL
LIN {X 0,Y 130.605,Z 816.879,A -85,B 0,C 180,E1 22963.4,E2 22963.4} C_VEL
LIN {X 0,Y 134.346,Z 808.564,A -85,B 0,C 180,E1 22978.61,E2 22978.61} C_VEL
LIN {X 0,Y 145.775,Z 794.801,A -85,B 0,C 180,E1 22992.164,E2 22992.164} C_VEL
LIN {X 0,Y 162.647,Z 776.303,A -85,B 0,C 180,E1 23002.598,E2 23002.598} C_VEL
LIN {X 0,Y 183.468,Z 751.464,A -85,B 0,C 180,E1 23010.657,E2 23010.657} C_VEL
LIN {X 0,Y 203.069,Z 723.867,A -85,B 0,C 180,E1 23015.78,E2 23015.78} C_VEL
LIN {X 0,Y 205.572,Z 719.67,A -85,B 0,C 180,E1 23016.459,E2 23016.459} C_VEL
LIN {X 0,Y 205.215,Z 704.176,A -85,B 0,C 180,E1 23023.543,E2 23023.543} C_VEL
LIN {X 0,Y 203.874,Z 693.633,A -85,B 0,C 180,E1 23030.416,E2 23030.416} C_VEL
LIN {X 0,Y 202.621,Z 686.632,A -85,B 0,C 180,E1 23037.871,E2 23037.871} C_VEL
LIN {X 0,Y 202.598,Z 685.113,A -85,B 0,C 180,E1 23040.012,E2 23040.012} C_VEL
LIN {X 0,Y 201.677,Z 684.878,A -85,B 0,C 180,E1 23044.317,E2 23044.317} C_VEL
LIN {X 0,Y 199.483,Z 690.971,A -85,B 0,C 180,E1 23054.358,E2 23054.358} C_VEL
LIN {X 0,Y 198.048,Z 699.582,A -85,B 0,C 180,E1 23061.747,E2 23061.747} C_VEL
LIN {X 0,Y 195.46,Z 711.611,A -85,B 0,C 180,E1 23069.308,E2 23069.308} C_VEL
LIN {X 0,Y 191.497,Z 723.889,A -85,B 0,C 180,E1 23075.924,E2 23075.924} C_VEL
LIN {X 0,Y 188.489,Z 728.248,A -85,B 0,C 180,E1 23077.522,E2 23077.522} C_VEL
LIN {X 0,Y 169.094,Z 749.065,A -85,B 0,C 180,E1 23085.415,E2 23085.415} C_VEL
LIN {X 0,Y 152.733,Z 763.776,A -85,B 0,C 180,E1 23095.257,E2 23095.257} C_VEL
LIN {X 0,Y 140.292,Z 773.814,A -85,B 0,C 180,E1 23107.814,E2 23107.814} C_VEL
LIN {X 0,Y 133.904,Z 778.821,A -85,B 0,C 180,E1 23123.514,E2 23123.514} C_VEL
LIN {X 0,Y 133.507,Z 778.943,A -85,B 0,C 180,E1 23134.703,E2 23134.703} C_VEL
LIN {X 0,Y 132.262,Z 778.548,A -85,B 0,C 180,E1 23140.33,E2 23140.33} C_VEL
LIN {X 0,Y 130.519,Z 776.754,A -85,B 0,C 180,E1 23149.425,E2 23149.425} C_VEL
LIN {X 0,Y 130.767,Z 776.529,A -85,B 0,C 180,E1 23149.891,E2 23149.891} C_VEL
LIN {X 0,Y 142.99,Z 767.523,A -85,B 0,C 180,E1 23163.778,E2 23163.778} C_VEL
LIN {X 0,Y 160.04,Z 753.35,A -85,B 0,C 180,E1 23174.708,E2 23174.708} C_VEL
LIN {X 0,Y 180.035,Z 733.54,A -85,B 0,C 180,E1 23183.034,E2 23183.034} C_VEL
LIN {X 0,Y 185.239,Z 727.287,A -85,B 0,C 180,E1 23185.085,E2 23185.085} C_VEL
LIN {X 0,Y 189.996,Z 714.949,A -85,B 0,C 180,E1 23192.078,E2 23192.078} C_VEL
LIN {X 0,Y 193.148,Z 703.195,A -85,B 0,C 180,E1 23200.171,E2 23200.171} C_VEL
LIN {X 0,Y 194.824,Z 696.533,A -85,B 0,C 180,E1 23206.505,E2 23206.505} C_VEL
LIN {X 0,Y 197.309,Z 691.381,A -85,B 0,C 180,E1 23216.032,E2 23216.032} C_VEL
LIN {X 0,Y 198.268,Z 691.618,A -85,B 0,C 180,E1 23219.988,E2 23219.988} C_VEL
LIN {X 0,Y 199.042,Z 699.102,A -85,B 0,C 180,E1 23228.738,E2 23228.738} C_VEL
LIN {X 0,Y 199.905,Z 709.907,A -85,B 0,C 180,E1 23236.023,E2 23236.023} C_VEL
LIN {X 0,Y 199.506,Z 722.739,A -85,B 0,C 180,E1 23242.148,E2 23242.148} C_VEL
LIN {X 0,Y 178.401,Z 751.501,A -85,B 0,C 180,E1 23247.443,E2 23247.443} C_VEL
LIN {X 0,Y 157.013,Z 775.639,A -85,B 0,C 180,E1 23255.331,E2 23255.331} C_VEL
LIN {X 0,Y 137.988,Z 795.3,A -85,B 0,C 180,E1 23266.995,E2 23266.995} C_VEL
LIN {X 0,Y 126.266,Z 808.401,A -85,B 0,C 180,E1 23281.332,E2 23281.332} C_VEL
LIN {X 0,Y 122.729,Z 815.618,A -85,B 0,C 180,E1 23295.709,E2 23295.709} C_VEL
LIN {X 0,Y 123.825,Z 818.365,A -85,B 0,C 180,E1 23309.994,E2 23309.994} C_VEL
LIN {X 0,Y 122.779,Z 815.655,A -85,B 0,C 180,E1 23324.271,E2 23324.271} C_VEL
LIN {X 0,Y 127.204,Z 807.317,A -85,B 0,C 180,E1 23340.38,E2 23340.38} C_VEL
LIN {X 0,Y 140.642,Z 792.673,A -85,B 0,C 180,E1 23355.066,E2 23355.066} C_VEL
LIN {X 0,Y 159.255,Z 773.505,A -85,B 0,C 180,E1 23365.62,E2 23365.62} C_VEL
LIN {X 0,Y 181.021,Z 748.361,A -85,B 0,C 180,E1 23373.342,E2 23373.342} C_VEL
LIN {X 0,Y 199.791,Z 722.671,A -85,B 0,C 180,E1 23377.877,E2 23377.877} C_VEL
LIN {X 0,Y 199.976,Z 707.625,A -85,B 0,C 180,E1 23385.384,E2 23385.384} C_VEL
LIN {X 0,Y 198.869,Z 696.968,A -85,B 0,C 180,E1 23393.455,E2 23393.455} C_VEL
LIN {X 0,Y 198.359,Z 691.924,A -85,B 0,C 180,E1 23400.012,E2 23400.012} C_VEL
LIN {X 0,Y 197.366,Z 691.656,A -85,B 0,C 180,E1 23404.412,E2 23404.412} C_VEL
LIN {X 0,Y 194.685,Z 697.799,A -85,B 0,C 180,E1 23414.653,E2 23414.653} C_VEL
LIN {X 0,Y 192.444,Z 706.89,A -85,B 0,C 180,E1 23422.379,E2 23422.379} C_VEL
LIN {X 0,Y 189.092,Z 718.08,A -85,B 0,C 180,E1 23429.57,E2 23429.57} C_VEL
LIN {X 0,Y 185.116,Z 727.954,A -85,B 0,C 180,E1 23435.135,E2 23435.135} C_VEL
LIN {X 0,Y 165.078,Z 748.92,A -85,B 0,C 180,E1 23442.808,E2 23442.808} C_VEL
LIN {X 0,Y 146.389,Z 764.965,A -85,B 0,C 180,E1 23453.516,E2 23453.516} C_VEL
LIN {X 0,Y 133.082,Z 775.004,A -85,B 0,C 180,E1 23466.542,E2 23466.542} C_VEL
LIN {X 0,Y 126.159,Z 780.005,A -85,B 0,C 180,E1 23483.114,E2 23483.114} C_VEL
LIN {X 0,Y 126.17,Z 779.974,A -85,B 0,C 180,E1 23496.898,E2 23496.898} C_VEL
LIN {X 0,Y 130.767,Z 776.529,A -85,B 0,C 180,E1 23509.891,E2 23509.891} C_VEL
LIN {X 0,Y 132.152,Z 773.704,A -85,B 0,C 180,E1 23517.418,E2 23517.418} C_VEL
LIN {X 0,Y 135.33,Z 769.584,A -85,B 0,C 180,E1 23524.611,E2 23524.611} C_VEL
LIN {X 0,Y 154.18,Z 754.908,A -85,B 0,C 180,E1 23536.554,E2 23536.554} C_VEL
LIN {X 0,Y 174.867,Z 735.362,A -85,B 0,C 180,E1 23544.877,E2 23544.877} C_VEL
LIN {X 0,Y 179.478,Z 730.19,A -85,B 0,C 180,E1 23546.567,E2 23546.567} C_VEL
LIN {X 0,Y 184.323,Z 719.432,A -85,B 0,C 180,E1 23553.053,E2 23553.053} C_VEL
LIN {X 0,Y 188.157,Z 708.337,A -85,B 0,C 180,E1 23561.211,E2 23561.211} C_VEL
LIN {X 0,Y 190.441,Z 701.563,A -85,B 0,C 180,E1 23568.523,E2 23568.523} C_VEL
LIN {X 0,Y 192.611,Z 698.198,A -85,B 0,C 180,E1 23575.479,E2 23575.479} C_VEL
LIN {X 0,Y 193.762,Z 698.25,A -85,B 0,C 180,E1 23579.988,E2 23579.988} C_VEL
LIN {X 0,Y 194.321,Z 705.944,A -85,B 0,C 180,E1 23588.952,E2 23588.952} C_VEL
LIN {X 0,Y 194.522,Z 717.107,A -85,B 0,C 180,E1 23596.375,E2 23596.375} C_VEL
LIN {X 0,Y 193.969,Z 725.297,A -85,B 0,C 180,E1 23600.491,E2 23600.491} C_VEL
LIN {X 0,Y 172.531,Z 752.803,A -85,B 0,C 180,E1 23605.722,E2 23605.722} C_VEL
LIN {X 0,Y 150.072,Z 776.758,A -85,B 0,C 180,E1 23613.863,E2 23613.863} C_VEL
LIN {X 0,Y 130.469,Z 795.526,A -85,B 0,C 180,E1 23625.863,E2 23625.863} C_VEL
LIN {X 0,Y 117.625,Z 809.091,A -85,B 0,C 180,E1 23642.59,E2 23642.59} C_VEL
LIN {X 0,Y 114.918,Z 814.391,A -85,B 0,C 180,E1 23654.715,E2 23654.715} C_VEL
LIN {X 0,Y 115.949,Z 817.168,A -85,B 0,C 180,E1 23669.993,E2 23669.993} C_VEL
LIN {X 0,Y 114.958,Z 814.427,A -85,B 0,C 180,E1 23685.265,E2 23685.265} C_VEL
LIN {X 0,Y 120.199,Z 806.07,A -85,B 0,C 180,E1 23702.358,E2 23702.358} C_VEL
LIN {X 0,Y 135.406,Z 790.958,A -85,B 0,C 180,E1 23717.889,E2 23717.889} C_VEL
LIN {X 0,Y 155.374,Z 771.629,A -85,B 0,C 180,E1 23728.388,E2 23728.388} C_VEL
LIN {X 0,Y 176.848,Z 747.882,A -85,B 0,C 180,E1 23735.513,E2 23735.513} C_VEL
LIN {X 0,Y 194.22,Z 724.742,A -85,B 0,C 180,E1 23739.804,E2 23739.804} C_VEL
LIN {X 0,Y 194.718,Z 712.323,A -85,B 0,C 180,E1 23746.523,E2 23746.523} C_VEL
LIN {X 0,Y 194.236,Z 703.761,A -85,B 0,C 180,E1 23753.298,E2 23753.298} C_VEL
LIN {X 0,Y 193.852,Z 698.555,A -85,B 0,C 180,E1 23760.012,E2 23760.012} C_VEL
LIN {X 0,Y 192.829,Z 698.323,A -85,B 0,C 180,E1 23764.516,E2 23764.516} C_VEL
LIN {X 0,Y 189.958,Z 703.583,A -85,B 0,C 180,E1 23773.847,E2 23773.847} C_VEL
LIN {X 0,Y 187.159,Z 711.836,A -85,B 0,C 180,E1 23781.412,E2 23781.412} C_VEL
LIN {X 0,Y 182.926,Z 723.243,A -85,B 0,C 180,E1 23789.141,E2 23789.141} C_VEL
LIN {X 0,Y 178.497,Z 731.734,A -85,B 0,C 180,E1 23793.867,E2 23793.867} C_VEL
LIN {X 0,Y 157.677,Z 752.034,A -85,B 0,C 180,E1 23801.746,E2 23801.746} C_VEL
LIN {X 0,Y 138.279,Z 767.594,A -85,B 0,C 180,E1 23812.98,E2 23812.98} C_VEL
LIN {X 0,Y 125.474,Z 776.501,A -85,B 0,C 180,E1 23825.784,E2 23825.784} C_VEL
LIN {X 0,Y 118.421,Z 781.19,A -85,B 0,C 180,E1 23842.661,E2 23842.661} C_VEL
LIN {X 0,Y 118.431,Z 781.159,A -85,B 0,C 180,E1 23857.352,E2 23857.352} C_VEL
LIN {X 0,Y 125.602,Z 776.365,A -85,B 0,C 180,E1 23874.323,E2 23874.323} C_VEL
LIN {X 0,Y 135.33,Z 769.584,A -85,B 0,C 180,E1 23884.611,E2 23884.611} C_VEL
LIN {X 0,Y 140.125,Z 764.506,A -85,B 0,C 180,E1 23891.292,E2 23891.292} C_VEL
LIN {X 0,Y 146.154,Z 758.264,A -85,B 0,C 180,E1 23897.412,E2 23897.412} C_VEL
LIN {X 0,Y 167.834,Z 739.281,A -85,B 0,C 180,E1 23906.136,E2 23906.136} C_VEL
LIN {X 0,Y 174.213,Z 732.423,A -85,B 0,C 180,E1 23908.555,E2 23908.555} C_VEL
LIN {X 0,Y 179.953,Z 720.878,A -85,B 0,C 180,E1 23916.159,E2 23916.159} C_VEL
LIN {X 0,Y 184.071,Z 711.049,A -85,B 0,C 180,E1 23924.589,E2 23924.589} C_VEL
LIN {X 0,Y 186.624,Z 705.877,A -85,B 0,C 180,E1 23932.552,E2 23932.552} C_VEL
LIN {X 0,Y 187.774,Z 704.692,A -85,B 0,C 180,E1 23935.362,E2 23935.362} C_VEL
LIN {X 0,Y 189.045,Z 704.729,A -85,B 0,C 180,E1 23939.987,E2 23939.987} C_VEL
LIN {X 0,Y 189.305,Z 711.333,A -85,B 0,C 180,E1 23948.033,E2 23948.033} C_VEL
LIN {X 0,Y 189.047,Z 721.154,A -85,B 0,C 180,E1 23955.074,E2 23955.074} C_VEL
LIN {X 0,Y 188.39,Z 727.823,A -85,B 0,C 180,E1 23958.738,E2 23958.738} C_VEL
LIN {X 0,Y 165.922,Z 755.11,A -85,B 0,C 180,E1 23964.137,E2 23964.137} C_VEL
LIN {X 0,Y 143.224,Z 777.722,A -85,B 0,C 180,E1 23972.245,E2 23972.245} C_VEL
LIN {X 0,Y 122.768,Z 795.994,A -85,B 0,C 180,E1 23984.828,E2 23984.828} C_VEL
LIN {X 0,Y 110.151,Z 808.158,A -85,B 0,C 180,E1 24001.236,E2 24001.236} C_VEL
LIN {X 0,Y 107.157,Z 813.166,A -85,B 0,C 180,E1 24013.578,E2 24013.578} C_VEL
LIN {X 0,Y 108.068,Z 815.971,A -85,B 0,C 180,E1 24029.993,E2 24029.993} C_VEL
LIN {X 0,Y 107.187,Z 813.201,A -85,B 0,C 180,E1 24046.402,E2 24046.402} C_VEL
LIN {X 0,Y 114.104,Z 804.023,A -85,B 0,C 180,E1 24065.725,E2 24065.725} C_VEL
LIN {X 0,Y 131.632,Z 788.29,A -85,B 0,C 180,E1 24081.635,E2 24081.635} C_VEL
LIN {X 0,Y 154.177,Z 767.458,A -85,B 0,C 180,E1 24092.093,E2 24092.093} C_VEL
LIN {X 0,Y 176.685,Z 742.988,A -85,B 0,C 180,E1 24098.717,E2 24098.717} C_VEL
LIN {X 0,Y 188.495,Z 727.979,A -85,B 0,C 180,E1 24101.273,E2 24101.273} C_VEL
LIN {X 0,Y 189.439,Z 715.833,A -85,B 0,C 180,E1 24108.488,E2 24108.488} C_VEL
LIN {X 0,Y 189.159,Z 708.316,A -85,B 0,C 180,E1 24115.422,E2 24115.422} C_VEL
LIN {X 0,Y 189.123,Z 705.021,A -85,B 0,C 180,E1 24120.013,E2 24120.013} C_VEL
LIN {X 0,Y 187.992,Z 704.812,A -85,B 0,C 180,E1 24124.632,E2 24124.632} C_VEL
LIN {X 0,Y 184.66,Z 710.223,A -85,B 0,C 180,E1 24134.253,E2 24134.253} C_VEL
LIN {X 0,Y 180.987,Z 718.822,A -85,B 0,C 180,E1 24142.062,E2 24142.062} C_VEL
LIN {X 0,Y 176.128,Z 729.279,A -85,B 0,C 180,E1 24149.293,E2 24149.293} C_VEL
LIN {X 0,Y 173.092,Z 734.228,A -85,B 0,C 180,E1 24152.105,E2 24152.105} C_VEL
LIN {X 0,Y 151.59,Z 754.047,A -85,B 0,C 180,E1 24159.983,E2 24159.983} C_VEL
LIN {X 0,Y 132.132,Z 768.784,A -85,B 0,C 180,E1 24170.942,E2 24170.942} C_VEL
LIN {X 0,Y 118.964,Z 777.336,A -85,B 0,C 180,E1 24183.453,E2 24183.453} C_VEL
LIN {X 0,Y 110.69,Z 782.374,A -85,B 0,C 180,E1 24202.146,E2 24202.146} C_VEL
LIN {X 0,Y 110.7,Z 782.344,A -85,B 0,C 180,E1 24217.868,E2 24217.868} C_VEL
LIN {X 0,Y 116.462,Z 778.751,A -85,B 0,C 180,E1 24232.962,E2 24232.962} C_VEL
LIN {X 0,Y 130.272,Z 769.908,A -85,B 0,C 180,E1 24247.608,E2 24247.608} C_VEL
LIN {X 0,Y 146.154,Z 758.264,A -85,B 0,C 180,E1 24257.412,E2 24257.412} C_VEL
LIN {X 0,Y 153.282,Z 751.038,A -85,B 0,C 180,E1 24262.912,E2 24262.912} C_VEL
LIN {X 0,Y 159.972,Z 743.856,A -85,B 0,C 180,E1 24267.233,E2 24267.233} C_VEL
LIN {X 0,Y 161.28,Z 742.642,A -85,B 0,C 180,E1 24267.687,E2 24267.687} C_VEL
LIN {X 0,Y 168.714,Z 735.33,A -85,B 0,C 180,E1 24270.277,E2 24270.277} C_VEL
LIN {X 0,Y 174.396,Z 725.371,A -85,B 0,C 180,E1 24277.248,E2 24277.248} C_VEL
LIN {X 0,Y 178.855,Z 716.574,A -85,B 0,C 180,E1 24285.274,E2 24285.274} C_VEL
LIN {X 0,Y 181.625,Z 712.088,A -85,B 0,C 180,E1 24292.731,E2 24292.731} C_VEL
LIN {X 0,Y 182.733,Z 711.032,A -85,B 0,C 180,E1 24295.234,E2 24295.234} C_VEL
LIN {X 0,Y 184.13,Z 711.068,A -85,B 0,C 180,E1 24299.987,E2 24299.987} C_VEL
LIN {X 0,Y 184.039,Z 718.023,A -85,B 0,C 180,E1 24308.384,E2 24308.384} C_VEL
LIN {X 0,Y 183.185,Z 727.86,A -85,B 0,C 180,E1 24315.381,E2 24315.381} C_VEL
LIN {X 0,Y 182.265,Z 731.347,A -85,B 0,C 180,E1 24317.086,E2 24317.086} C_VEL
LIN {X 0,Y 159.37,Z 757.293,A -85,B 0,C 180,E1 24322.427,E2 24322.427} C_VEL
LIN {X 0,Y 136.287,Z 778.815,A -85,B 0,C 180,E1 24330.565,E2 24330.565} C_VEL
LIN {X 0,Y 115.114,Z 796.391,A -85,B 0,C 180,E1 24343.656,E2 24343.656} C_VEL
LIN {X 0,Y 103.072,Z 806.918,A -85,B 0,C 180,E1 24359.053,E2 24359.053} C_VEL
LIN {X 0,Y 99.405,Z 811.934,A -85,B 0,C 180,E1 24372.256,E2 24372.256} C_VEL
LIN {X 0,Y 100.183,Z 814.773,A -85,B 0,C 180,E1 24389.992,E2 24389.992} C_VEL
LIN {X 0,Y 99.431,Z 811.969,A -85,B 0,C 180,E1 24407.722,E2 24407.722} C_VEL
LIN {X 0,Y 107.367,Z 802.929,A -85,B 0,C 180,E1 24428.051,E2 24428.051} C_VEL
LIN {X 0,Y 124.982,Z 788.393,A -85,B 0,C 180,E1 24443.549,E2 24443.549} C_VEL
LIN {X 0,Y 147.553,Z 769,A -85,B 0,C 180,E1 24453.861,E2 24453.861} C_VEL
LIN {X 0,Y 172.271,Z 743.541,A -85,B 0,C 180,E1 24460.855,E2 24460.855} C_VEL
LIN {X 0,Y 181.993,Z 732.014,A -85,B 0,C 180,E1 24462.843,E2 24462.843} C_VEL
LIN {X 0,Y 183.204,Z 728.714,A -85,B 0,C 180,E1 24464.217,E2 24464.217} C_VEL
LIN {X 0,Y 184.154,Z 718.219,A -85,B 0,C 180,E1 24471.621,E2 24471.621} C_VEL
LIN {X 0,Y 184.194,Z 711.351,A -85,B 0,C 180,E1 24480.013,E2 24480.013} C_VEL
LIN {X 0,Y 182.548,Z 711.487,A -85,B 0,C 180,E1 24485.627,E2 24485.627} C_VEL
LIN {X 0,Y 178.965,Z 716.814,A -85,B 0,C 180,E1 24494.716,E2 24494.716} C_VEL
LIN {X 0,Y 174.429,Z 725.68,A -85,B 0,C 180,E1 24502.783,E2 24502.783} C_VEL
LIN {X 0,Y 168.795,Z 735.533,A -85,B 0,C 180,E1 24509.699,E2 24509.699} C_VEL
LIN {X 0,Y 147.236,Z 754.815,A -85,B 0,C 180,E1 24517.414,E2 24517.414} C_VEL
LIN {X 0,Y 126.154,Z 769.976,A -85,B 0,C 180,E1 24528.703,E2 24528.703} C_VEL
LIN {X 0,Y 112.011,Z 778.527,A -85,B 0,C 180,E1 24541.662,E2 24541.662} C_VEL
LIN {X 0,Y 102.969,Z 783.558,A -85,B 0,C 180,E1 24561.553,E2 24561.553} C_VEL
LIN {X 0,Y 102.98,Z 783.529,A -85,B 0,C 180,E1 24578.462,E2 24578.462} C_VEL
LIN {X 0,Y 112.248,Z 778.304,A -85,B 0,C 180,E1 24598.577,E2 24598.577} C_VEL
LIN {X 0,Y 128.316,Z 768.377,A -85,B 0,C 180,E1 24612.731,E2 24612.731} C_VEL
LIN {X 0,Y 150.231,Z 752.27,A -85,B 0,C 180,E1 24623.739,E2 24623.739} C_VEL
LIN {X 0,Y 161.28,Z 742.642,A -85,B 0,C 180,E1 24627.687,E2 24627.687} C_VEL
LIN {X 0,Y 164.37,Z 738.725,A -85,B 0,C 180,E1 24630.129,E2 24630.129} C_VEL
LIN {X 0,Y 166.216,Z 733.859,A -85,B 0,C 180,E1 24635.199,E2 24635.199} C_VEL
LIN {X 0,Y 171.496,Z 725.379,A -85,B 0,C 180,E1 24642.401,E2 24642.401} C_VEL
LIN {X 0,Y 175.407,Z 719.278,A -85,B 0,C 180,E1 24650.045,E2 24650.045} C_VEL
LIN {X 0,Y 177.469,Z 717.25,A -85,B 0,C 180,E1 24655.092,E2 24655.092} C_VEL
LIN {X 0,Y 179.043,Z 717.237,A -85,B 0,C 180,E1 24659.986,E2 24659.986} C_VEL
LIN {X 0,Y 178.689,Z 722.942,A -85,B 0,C 180,E1 24667.291,E2 24667.291} C_VEL
LIN {X 0,Y 177.503,Z 731.967,A -85,B 0,C 180,E1 24674.181,E2 24674.181} C_VEL
LIN {X 0,Y 176.797,Z 733.923,A -85,B 0,C 180,E1 24675.189,E2 24675.189} C_VEL
LIN {X 0,Y 151.762,Z 760.52,A -85,B 0,C 180,E1 24680.879,E2 24680.879} C_VEL
LIN {X 0,Y 126.396,Z 782.286,A -85,B 0,C 180,E1 24690.134,E2 24690.134} C_VEL
LIN {X 0,Y 105.507,Z 798.182,A -85,B 0,C 180,E1 24704.141,E2 24704.141} C_VEL
LIN {X 0,Y 94.095,Z 807.59,A -85,B 0,C 180,E1 24721.128,E2 24721.128} C_VEL
LIN {X 0,Y 91.287,Z 812.68,A -85,B 0,C 180,E1 24740.444,E2 24740.444} C_VEL
LIN {X 0,Y 92.287,Z 813.574,A -85,B 0,C 180,E1 24749.991,E2 24749.991} C_VEL
LIN {X 0,Y 91.724,Z 810.735,A -85,B 0,C 180,E1 24769.267,E2 24769.267} C_VEL
LIN {X 0,Y 100.29,Z 802.285,A -85,B 0,C 180,E1 24789.983,E2 24789.983} C_VEL
LIN {X 0,Y 120.606,Z 786.918,A -85,B 0,C 180,E1 24806.851,E2 24806.851} C_VEL
LIN {X 0,Y 145.673,Z 766.333,A -85,B 0,C 180,E1 24817.266,E2 24817.266} C_VEL
LIN {X 0,Y 169.778,Z 742.249,A -85,B 0,C 180,E1 24823.449,E2 24823.449} C_VEL
LIN {X 0,Y 177.402,Z 733.142,A -85,B 0,C 180,E1 24825.179,E2 24825.179} C_VEL
LIN {X 0,Y 178.688,Z 724.576,A -85,B 0,C 180,E1 24831.363,E2 24831.363} C_VEL
LIN {X 0,Y 178.917,Z 719.113,A -85,B 0,C 180,E1 24837.589,E2 24837.589} C_VEL
LIN {X 0,Y 179.086,Z 717.522,A -85,B 0,C 180,E1 24840.014,E2 24840.014} C_VEL
LIN {X 0,Y 177.7,Z 717.335,A -85,B 0,C 180,E1 24844.901,E2 24844.901} C_VEL
LIN {X 0,Y 174,Z 721.667,A -85,B 0,C 180,E1 24853.272,E2 24853.272} C_VEL
LIN {X 0,Y 169.268,Z 729.34,A -85,B 0,C 180,E1 24860.979,E2 24860.979} C_VEL
LIN {X 0,Y 163.69,Z 737.92,A -85,B 0,C 180,E1 24867.563,E2 24867.563} C_VEL
LIN {X 0,Y 149.875,Z 750.302,A -85,B 0,C 180,E1 24872.227,E2 24872.227} C_VEL
LIN {X 0,Y 127.225,Z 766.831,A -85,B 0,C 180,E1 24882.052,E2 24882.052} C_VEL
LIN {X 0,Y 108.441,Z 777.973,A -85,B 0,C 180,E1 24896.059,E2 24896.059} C_VEL
LIN {X 0,Y 97.804,Z 783.475,A -85,B 0,C 180,E1 24911.973,E2 24911.973} C_VEL
LIN {X 0,Y 94.045,Z 785.268,A -85,B 0,C 180,E1 24930.009,E2 24930.009} C_VEL
LIN {X 0,Y 97.822,Z 783.427,A -85,B 0,C 180,E1 24948.04,E2 24948.04} C_VEL
LIN {X 0,Y 110.248,Z 776.898,A -85,B 0,C 180,E1 24965.716,E2 24965.716} C_VEL
LIN {X 0,Y 129.854,Z 764.942,A -85,B 0,C 180,E1 24979.285,E2 24979.285} C_VEL
LIN {X 0,Y 152.846,Z 747.682,A -85,B 0,C 180,E1 24988.698,E2 24988.698} C_VEL
LIN {X 0,Y 162.503,Z 739.034,A -85,B 0,C 180,E1 24991.661,E2 24991.661} C_VEL
LIN {X 0,Y 166.216,Z 733.859,A -85,B 0,C 180,E1 24995.199,E2 24995.199} C_VEL
LIN {X 0,Y 167.736,Z 730.296,A -85,B 0,C 180,E1 24999.49,E2 24999.49} C_VEL
LIN {X 0,Y 168.316,Z 727.071,A -85,B 0,C 180,E1 25007.104,E2 25007.104} C_VEL
LIN {X 0,Y 172.019,Z 723.292,A -85,B 0,C 180,E1 25014.936,E2 25014.936} C_VEL
LIN {X 0,Y 173.673,Z 723.211,A -85,B 0,C 180,E1 25019.986,E2 25019.986} C_VEL
LIN {X 0,Y 173.042,Z 729.171,A -85,B 0,C 180,E1 25027.527,E2 25027.527} C_VEL
LIN {X 0,Y 171.923,Z 735.137,A -85,B 0,C 180,E1 25032.376,E2 25032.376} C_VEL
LIN {X 0,Y 171.109,Z 736.914,A -85,B 0,C 180,E1 25033.247,E2 25033.247} C_VEL
LIN {X 0,Y 145.918,Z 762.006,A -85,B 0,C 180,E1 25038.751,E2 25038.751} C_VEL
LIN {X 0,Y 119.981,Z 782.896,A -85,B 0,C 180,E1 25047.941,E2 25047.941} C_VEL
LIN {X 0,Y 97.923,Z 798.294,A -85,B 0,C 180,E1 25062.643,E2 25062.643} C_VEL
LIN {X 0,Y 85.759,Z 807.503,A -85,B 0,C 180,E1 25081.913,E2 25081.913} C_VEL
LIN {X 0,Y 83.386,Z 811.461,A -85,B 0,C 180,E1 25099.529,E2 25099.529} C_VEL
LIN {X 0,Y 84.409,Z 812.377,A -85,B 0,C 180,E1 25109.991,E2 25109.991} C_VEL
LIN {X 0,Y 84.099,Z 809.502,A -85,B 0,C 180,E1 25131.093,E2 25131.093} C_VEL
LIN {X 0,Y 94.138,Z 801.035,A -85,B 0,C 180,E1 25153.2,E2 25153.2} C_VEL
LIN {X 0,Y 115.41,Z 786.301,A -85,B 0,C 180,E1 25169.776,E2 25169.776} C_VEL
LIN {X 0,Y 141.11,Z 766.471,A -85,B 0,C 180,E1 25179.837,E2 25179.837} C_VEL
LIN {X 0,Y 165.922,Z 742.796,A -85,B 0,C 180,E1 25185.797,E2 25185.797} C_VEL
LIN {X 0,Y 171.092,Z 737.219,A -85,B 0,C 180,E1 25186.736,E2 25186.736} C_VEL
LIN {X 0,Y 172.68,Z 732.232,A -85,B 0,C 180,E1 25189.915,E2 25189.915} C_VEL
LIN {X 0,Y 173.535,Z 725.104,A -85,B 0,C 180,E1 25197.514,E2 25197.514} C_VEL
LIN {X 0,Y 173.715,Z 723.494,A -85,B 0,C 180,E1 25200.014,E2 25200.014} C_VEL
LIN {X 0,Y 172.208,Z 723.414,A -85,B 0,C 180,E1 25205.058,E2 25205.058} C_VEL
LIN {X 0,Y 168.325,Z 727.41,A -85,B 0,C 180,E1 25213.007,E2 25213.007} C_VEL
LIN {X 0,Y 163.55,Z 733.942,A -85,B 0,C 180,E1 25219.984,E2 25219.984} C_VEL
LIN {X 0,Y 157.543,Z 741.752,A -85,B 0,C 180,E1 25226.179,E2 25226.179} C_VEL
LIN {X 0,Y 132.932,Z 761.009,A -85,B 0,C 180,E1 25234.348,E2 25234.348} C_VEL
LIN {X 0,Y 110.215,Z 774.884,A -85,B 0,C 180,E1 25246.629,E2 25246.629} C_VEL
LIN {X 0,Y 92.571,Z 783.638,A -85,B 0,C 180,E1 25265.875,E2 25265.875} C_VEL
LIN {X 0,Y 87.573,Z 785.927,A -85,B 0,C 180,E1 25280.054,E2 25280.054} C_VEL
LIN {X 0,Y 87.583,Z 785.899,A -85,B 0,C 180,E1 25299.964,E2 25299.964} C_VEL
LIN {X 0,Y 98.372,Z 780.918,A -85,B 0,C 180,E1 25322.378,E2 25322.378} C_VEL
LIN {X 0,Y 117.296,Z 770.77,A -85,B 0,C 180,E1 25337.929,E2 25337.929} C_VEL
LIN {X 0,Y 141.549,Z 754.687,A -85,B 0,C 180,E1 25348.846,E2 25348.846} C_VEL
LIN {X 0,Y 157.585,Z 741.496,A -85,B 0,C 180,E1 25353.755,E2 25353.755} C_VEL
LIN {X 0,Y 163.554,Z 733.648,A -85,B 0,C 180,E1 25360.041,E2 25360.041} C_VEL
LIN {X 0,Y 168.316,Z 727.071,A -85,B 0,C 180,E1 25367.104,E2 25367.104} C_VEL
LIN {X 0,Y 168.497,Z 726.501,A -85,B 0,C 180,E1 25371.558,E2 25371.558} C_VEL
LIN {X 0,Y 167.779,Z 729,A -85,B 0,C 180,E1 25379.203,E2 25379.203} C_VEL
LIN {X 0,Y 167.487,Z 733.439,A -85,B 0,C 180,E1 25386.046,E2 25386.046} C_VEL
LIN {X 0,Y 165.863,Z 739.434,A -85,B 0,C 180,E1 25391.159,E2 25391.159} C_VEL
LIN {X 0,Y 140.155,Z 763.572,A -85,B 0,C 180,E1 25396.501,E2 25396.501} C_VEL
LIN {X 0,Y 113.419,Z 783.67,A -85,B 0,C 180,E1 25405.687,E2 25405.687} C_VEL
LIN {X 0,Y 91.021,Z 797.972,A -85,B 0,C 180,E1 25420.331,E2 25420.331} C_VEL
LIN {X 0,Y 78.661,Z 806.264,A -85,B 0,C 180,E1 25439.116,E2 25439.116} C_VEL
LIN {X 0,Y 75.498,Z 810.24,A -85,B 0,C 180,E1 25458.421,E2 25458.421} C_VEL
LIN {X 0,Y 76.492,Z 811.174,A -85,B 0,C 180,E1 25469.99,E2 25469.99} C_VEL
LIN {X 0,Y 76.561,Z 808.266,A -85,B 0,C 180,E1 25493.286,E2 25493.286} C_VEL
LIN {X 0,Y 88.08,Z 799.929,A -85,B 0,C 180,E1 25516.6,E2 25516.6} C_VEL
LIN {X 0,Y 110.5,Z 785.718,A -85,B 0,C 180,E1 25532.932,E2 25532.932} C_VEL
LIN {X 0,Y 136.853,Z 766.513,A -85,B 0,C 180,E1 25542.572,E2 25542.572} C_VEL
LIN {X 0,Y 162.907,Z 742.767,A -85,B 0,C 180,E1 25548.347,E2 25548.347} C_VEL
LIN {X 0,Y 166.485,Z 738.474,A -85,B 0,C 180,E1 25549.535,E2 25549.535} C_VEL
LIN {X 0,Y 167.69,Z 732.859,A -85,B 0,C 180,E1 25554.834,E2 25554.834} C_VEL
LIN {X 0,Y 168.147,Z 729.281,A -85,B 0,C 180,E1 25560.014,E2 25560.014} C_VEL
LIN {X 0,Y 166.441,Z 729.29,A -85,B 0,C 180,E1 25565.234,E2 25565.234} C_VEL
LIN {X 0,Y 161.914,Z 733.522,A -85,B 0,C 180,E1 25573.535,E2 25573.535} C_VEL
LIN {X 0,Y 155.59,Z 741.009,A -85,B 0,C 180,E1 25581.259,E2 25581.259} C_VEL
LIN {X 0,Y 152.416,Z 744.592,A -85,B 0,C 180,E1 25584.05,E2 25584.05} C_VEL
LIN {X 0,Y 128.682,Z 762.203,A -85,B 0,C 180,E1 25591.472,E2 25591.472} C_VEL
LIN {X 0,Y 104.667,Z 776.073,A -85,B 0,C 180,E1 25603.687,E2 25603.687} C_VEL
LIN {X 0,Y 88.504,Z 783.583,A -85,B 0,C 180,E1 25619.133,E2 25619.133} C_VEL
LIN {X 0,Y 79.899,Z 787.111,A -85,B 0,C 180,E1 25639.087,E2 25639.087} C_VEL
LIN {X 0,Y 79.91,Z 787.084,A -85,B 0,C 180,E1 25660.932,E2 25660.932} C_VEL
LIN {X 0,Y 91.656,Z 782.202,A -85,B 0,C 180,E1 25684.753,E2 25684.753} C_VEL
LIN {X 0,Y 112.207,Z 771.965,A -85,B 0,C 180,E1 25700.894,E2 25700.894} C_VEL
LIN {X 0,Y 137.674,Z 755.892,A -85,B 0,C 180,E1 25711.627,E2 25711.627} C_VEL
LIN {X 0,Y 152.526,Z 744.281,A -85,B 0,C 180,E1 25715.881,E2 25715.881} C_VEL
LIN {X 0,Y 158.832,Z 736.841,A -85,B 0,C 180,E1 25722.422,E2 25722.422} C_VEL
LIN {X 0,Y 163.626,Z 731.302,A -85,B 0,C 180,E1 25729.32,E2 25729.32} C_VEL
LIN {X 0,Y 166.87,Z 728.952,A -85,B 0,C 180,E1 25736.482,E2 25736.482} C_VEL
LIN {X 0,Y 167.779,Z 729,A -85,B 0,C 180,E1 25739.203,E2 25739.203} C_VEL
LIN {X 0,Y 166.419,Z 731.769,A -85,B 0,C 180,E1 25741.934,E2 25741.934} C_VEL
LIN {X 0,Y 161.407,Z 739.28,A -85,B 0,C 180,E1 25746.303,E2 25746.303} C_VEL
LIN {X 0,Y 160.238,Z 742.488,A -85,B 0,C 180,E1 25749.032,E2 25749.032} C_VEL
LIN {X 0,Y 132.938,Z 766.346,A -85,B 0,C 180,E1 25754.496,E2 25754.496} C_VEL
LIN {X 0,Y 107.027,Z 784.328,A -85,B 0,C 180,E1 25763.128,E2 25763.128} C_VEL
LIN {X 0,Y 82.654,Z 798.606,A -85,B 0,C 180,E1 25779.241,E2 25779.241} C_VEL
LIN {X 0,Y 69.145,Z 806.994,A -85,B 0,C 180,E1 25804.016,E2 25804.016} C_VEL
LIN {X 0,Y 68.607,Z 809.977,A -85,B 0,C 180,E1 25829.988,E2 25829.988} C_VEL
LIN {X 0,Y 69.157,Z 807.03,A -85,B 0,C 180,E1 25855.954,E2 25855.954} C_VEL
LIN {X 0,Y 82.645,Z 798.679,A -85,B 0,C 180,E1 25880.747,E2 25880.747} C_VEL
LIN {X 0,Y 107.007,Z 784.462,A -85,B 0,C 180,E1 25896.859,E2 25896.859} C_VEL
LIN {X 0,Y 134.612,Z 765.243,A -85,B 0,C 180,E1 25905.923,E2 25905.923} C_VEL
LIN {X 0,Y 160.237,Z 742.736,A -85,B 0,C 180,E1 25910.978,E2 25910.978} C_VEL
LIN {X 0,Y 161.92,Z 737.511,A -85,B 0,C 180,E1 25915.994,E2 25915.994} C_VEL
LIN {X 0,Y 162.415,Z 734.888,A -85,B 0,C 180,E1 25920.015,E2 25920.015} C_VEL
LIN {X 0,Y 160.454,Z 734.977,A -85,B 0,C 180,E1 25925.43,E2 25925.43} C_VEL
LIN {X 0,Y 155.624,Z 739.009,A -85,B 0,C 180,E1 25933.399,E2 25933.399} C_VEL
LIN {X 0,Y 148.624,Z 746.296,A -85,B 0,C 180,E1 25941.064,E2 25941.064} C_VEL
LIN {X 0,Y 137.218,Z 755.053,A -85,B 0,C 180,E1 25944.471,E2 25944.471} C_VEL
LIN {X 0,Y 110.153,Z 771.87,A -85,B 0,C 180,E1 25954.456,E2 25954.456} C_VEL
LIN {X 0,Y 89.934,Z 781.534,A -85,B 0,C 180,E1 25967.683,E2 25967.683} C_VEL
LIN {X 0,Y 75.844,Z 787.035,A -85,B 0,C 180,E1 25986.481,E2 25986.481} C_VEL
LIN {X 0,Y 70.617,Z 788.827,A -85,B 0,C 180,E1 26010.011,E2 26010.011} C_VEL
LIN {X 0,Y 75.869,Z 786.99,A -85,B 0,C 180,E1 26033.534,E2 26033.534} C_VEL
LIN {X 0,Y 92.226,Z 780.472,A -85,B 0,C 180,E1 26054.255,E2 26054.255} C_VEL
LIN {X 0,Y 117.129,Z 767.856,A -85,B 0,C 180,E1 26068.599,E2 26068.599} C_VEL
LIN {X 0,Y 143.721,Z 750.05,A -85,B 0,C 180,E1 26077.199,E2 26077.199} C_VEL
LIN {X 0,Y 148.645,Z 746.041,A -85,B 0,C 180,E1 26078.946,E2 26078.946} C_VEL
LIN {X 0,Y 155.642,Z 738.721,A -85,B 0,C 180,E1 26086.618,E2 26086.618} C_VEL
LIN {X 0,Y 160.344,Z 734.795,A -85,B 0,C 180,E1 26094.567,E2 26094.567} C_VEL
LIN {X 0,Y 162.388,Z 734.639,A -85,B 0,C 180,E1 26099.985,E2 26099.985} C_VEL
LIN {X 0,Y 161.407,Z 739.28,A -85,B 0,C 180,E1 26106.303,E2 26106.303} C_VEL
LIN {X 0,Y 158.477,Z 742.936,A -85,B 0,C 180,E1 26107.66,E2 26107.66} C_VEL
LIN {X 0,Y 144.274,Z 754.646,A -85,B 0,C 180,E1 26108.429,E2 26108.429} C_VEL
LIN {X 0,Y 114.401,Z 776.661,A -85,B 0,C 180,E1 26115.326,E2 26115.326} C_VEL
LIN {X 0,Y 85.901,Z 793.161,A -85,B 0,C 180,E1 26128.186,E2 26128.186} C_VEL
LIN {X 0,Y 65.333,Z 803.683,A -85,B 0,C 180,E1 26151.316,E2 26151.316} C_VEL
LIN {X 0,Y 59.816,Z 807.794,A -85,B 0,C 180,E1 26175.324,E2 26175.324} C_VEL
LIN {X 0,Y 60.526,Z 808.738,A -85,B 0,C 180,E1 26190.875,E2 26190.875} C_VEL
LIN {X 0,Y 61.959,Z 805.798,A -85,B 0,C 180,E1 26219.241,E2 26219.241} C_VEL
LIN {X 0,Y 80.506,Z 796.001,A -85,B 0,C 180,E1 26247.791,E2 26247.791} C_VEL
LIN {X 0,Y 108.924,Z 780.32,A -85,B 0,C 180,E1 26262.839,E2 26262.839} C_VEL
LIN {X 0,Y 138.173,Z 759.835,A -85,B 0,C 180,E1 26270.424,E2 26270.424} C_VEL
LIN {X 0,Y 153.51,Z 746.736,A -85,B 0,C 180,E1 26273.065,E2 26273.065} C_VEL
LIN {X 0,Y 155.52,Z 744.163,A -85,B 0,C 180,E1 26274.429,E2 26274.429} C_VEL
LIN {X 0,Y 156.502,Z 740.334,A -85,B 0,C 180,E1 26280.015,E2 26280.015} C_VEL
LIN {X 0,Y 154.252,Z 740.502,A -85,B 0,C 180,E1 26285.649,E2 26285.649} C_VEL
LIN {X 0,Y 150.437,Z 743.266,A -85,B 0,C 180,E1 26291.628,E2 26291.628} C_VEL
LIN {X 0,Y 143.813,Z 749.146,A -85,B 0,C 180,E1 26298.667,E2 26298.667} C_VEL
LIN {X 0,Y 137.465,Z 753.96,A -85,B 0,C 180,E1 26300.597,E2 26300.597} C_VEL
LIN {X 0,Y 109.111,Z 771.423,A -85,B 0,C 180,E1 26309.567,E2 26309.567} C_VEL
LIN {X 0,Y 84.307,Z 782.723,A -85,B 0,C 180,E1 26324.096,E2 26324.096} C_VEL
LIN {X 0,Y 68.749,Z 788.221,A -85,B 0,C 180,E1 26343.88,E2 26343.88} C_VEL
LIN {X 0,Y 62.807,Z 790.013,A -85,B 0,C 180,E1 26370.013,E2 26370.013} C_VEL
LIN {X 0,Y 68.776,Z 788.176,A -85,B 0,C 180,E1 26396.134,E2 26396.134} C_VEL
LIN {X 0,Y 89.335,Z 780.594,A -85,B 0,C 180,E1 26419.712,E2 26419.712} C_VEL
LIN {X 0,Y 115.391,Z 767.896,A -85,B 0,C 180,E1 26432.777,E2 26432.777} C_VEL
LIN {X 0,Y 143,Z 749.634,A -85,B 0,C 180,E1 26440.684,E2 26440.684} C_VEL
LIN {X 0,Y 148.407,Z 744.737,A -85,B 0,C 180,E1 26445.952,E2 26445.952} C_VEL
LIN {X 0,Y 152.883,Z 741.07,A -85,B 0,C 180,E1 26452.055,E2 26452.055} C_VEL
LIN {X 0,Y 156.479,Z 740.101,A -85,B 0,C 180,E1 26459.985,E2 26459.985} C_VEL
LIN {X 0,Y 155.188,Z 744.667,A -85,B 0,C 180,E1 26466.277,E2 26466.277} C_VEL
LIN {X 0,Y 148.958,Z 750.643,A -85,B 0,C 180,E1 26467.653,E2 26467.653} C_VEL
LIN {X 0,Y 144.274,Z 754.646,A -85,B 0,C 180,E1 26468.429,E2 26468.429} C_VEL
LIN {X 0,Y 130.061,Z 764.707,A -85,B 0,C 180,E1 26469.349,E2 26469.349} C_VEL
LIN {X 0,Y 115.222,Z 773.725,A -85,B 0,C 180,E1 26470.557,E2 26470.557} C_VEL
LIN {X 0,Y 85.166,Z 790.511,A -85,B 0,C 180,E1 26481.581,E2 26481.581} C_VEL
LIN {X 0,Y 61.483,Z 801.357,A -85,B 0,C 180,E1 26502.355,E2 26502.355} C_VEL
LIN {X 0,Y 52.069,Z 806.572,A -85,B 0,C 180,E1 26533.08,E2 26533.08} C_VEL
LIN {X 0,Y 52.741,Z 807.566,A -85,B 0,C 180,E1 26549.985,E2 26549.985} C_VEL
LIN {X 0,Y 55.565,Z 804.27,A -85,B 0,C 180,E1 26585.246,E2 26585.246} C_VEL
LIN {X 0,Y 76.432,Z 794.749,A -85,B 0,C 180,E1 26613.026,E2 26613.026} C_VEL
LIN {X 0,Y 106.785,Z 779.061,A -85,B 0,C 180,E1 26627.063,E2 26627.063} C_VEL
LIN {X 0,Y 137.044,Z 758.56,A -85,B 0,C 180,E1 26633.82,E2 26633.82} C_VEL
LIN {X 0,Y 148.061,Z 749.602,A -85,B 0,C 180,E1 26635.489,E2 26635.489} C_VEL
LIN {X 0,Y 149.668,Z 747.978,A -85,B 0,C 180,E1 26636.173,E2 26636.173} C_VEL
LIN {X 0,Y 150.37,Z 745.528,A -85,B 0,C 180,E1 26640.016,E2 26640.016} C_VEL
LIN {X 0,Y 147.853,Z 745.837,A -85,B 0,C 180,E1 26645.894,E2 26645.894} C_VEL
LIN {X 0,Y 143.148,Z 749.002,A -85,B 0,C 180,E1 26652.23,E2 26652.23} C_VEL
LIN {X 0,Y 138.015,Z 752.986,A -85,B 0,C 180,E1 26656.794,E2 26656.794} C_VEL
LIN {X 0,Y 108.557,Z 771.018,A -85,B 0,C 180,E1 26664.759,E2 26664.759} C_VEL
LIN {X 0,Y 81.693,Z 782.969,A -85,B 0,C 180,E1 26678.049,E2 26678.049} C_VEL
LIN {X 0,Y 61.83,Z 789.407,A -85,B 0,C 180,E1 26700.692,E2 26700.692} C_VEL
LIN {X 0,Y 54.998,Z 791.2,A -85,B 0,C 180,E1 26730.015,E2 26730.015} C_VEL
LIN {X 0,Y 61.859,Z 789.363,A -85,B 0,C 180,E1 26759.323,E2 26759.323} C_VEL
LIN {X 0,Y 84.491,Z 781.783,A -85,B 0,C 180,E1 26783.758,E2 26783.758} C_VEL
LIN {X 0,Y 112.918,Z 768.596,A -85,B 0,C 180,E1 26796.611,E2 26796.611} C_VEL
LIN {X 0,Y 138.113,Z 752.705,A -85,B 0,C 180,E1 26803.115,E2 26803.115} C_VEL
LIN {X 0,Y 144.846,Z 747.446,A -85,B 0,C 180,E1 26809.769,E2 26809.769} C_VEL
LIN {X 0,Y 147.975,Z 745.603,A -85,B 0,C 180,E1 26814.629,E2 26814.629} C_VEL
LIN {X 0,Y 150.331,Z 745.314,A -85,B 0,C 180,E1 26819.984,E2 26819.984} C_VEL
LIN {X 0,Y 149.648,Z 747.676,A -85,B 0,C 180,E1 26823.682,E2 26823.682} C_VEL
LIN {X 0,Y 146.248,Z 750.912,A -85,B 0,C 180,E1 26824.784,E2 26824.784} C_VEL
LIN {X 0,Y 117.53,Z 772.221,A -85,B 0,C 180,E1 26830.03,E2 26830.03} C_VEL
LIN {X 0,Y 115.222,Z 773.725,A -85,B 0,C 180,E1 26830.557,E2 26830.557} C_VEL
LIN {X 0,Y 99.916,Z 781.699,A -85,B 0,C 180,E1 26832.392,E2 26832.392} C_VEL
LIN {X 0,Y 84.426,Z 788.358,A -85,B 0,C 180,E1 26835.358,E2 26835.358} C_VEL
LIN {X 0,Y 56.282,Z 800.109,A -85,B 0,C 180,E1 26856.17,E2 26856.17} C_VEL
LIN {X 0,Y 44.4,Z 805.344,A -85,B 0,C 180,E1 26890.044,E2 26890.044} C_VEL
LIN {X 0,Y 44.792,Z 806.359,A -85,B 0,C 180,E1 26909.982,E2 26909.982} C_VEL
LIN {X 0,Y 48.377,Z 803.32,A -85,B 0,C 180,E1 26948.729,E2 26948.729} C_VEL
LIN {X 0,Y 73.071,Z 793.498,A -85,B 0,C 180,E1 26978.781,E2 26978.781} C_VEL
LIN {X 0,Y 105.258,Z 777.812,A -85,B 0,C 180,E1 26991.401,E2 26991.401} C_VEL
LIN {X 0,Y 136.405,Z 757.293,A -85,B 0,C 180,E1 26997.244,E2 26997.244} C_VEL
LIN {X 0,Y 142.116,Z 752.868,A -85,B 0,C 180,E1 26997.999,E2 26997.999} C_VEL
LIN {X 0,Y 144.049,Z 750.53,A -85,B 0,C 180,E1 27000.017,E2 27000.017} C_VEL
